	VAR robtarget Openhole_4144 := [[463.64, -19.43, 181.36], [0.050906, 0.705272, 0.70561, -0.045991], [0,0,0,0], [9E9, 9E9, 9E9, 9E9, 9E9, 9E9]];
	VAR robtarget Openhole_4145 := [[462.64, -19.54, 181.37], [0.047948, 0.705479, 0.70584, -0.042314], [0,0,0,0], [9E9, 9E9, 9E9, 9E9, 9E9, 9E9]];
	VAR robtarget Openhole_4146 := [[462.15, -19.58, 181.37], [0.046425, 0.705581, 0.705946, -0.040505], [0,0,0,0], [9E9, 9E9, 9E9, 9E9, 9E9, 9E9]];
	VAR robtarget Openhole_4147 := [[461.97, -18.21, 181.2], [0.041221, 0.705904, 0.705703, -0.044533], [0,0,0,0], [9E9, 9E9, 9E9, 9E9, 9E9, 9E9]];
	VAR robtarget Openhole_4148 := [[462.42, -18, 181.17], [0.042026, 0.705857, 0.705559, -0.046754], [0,0,0,0], [9E9, 9E9, 9E9, 9E9, 9E9, 9E9]];
	VAR robtarget Openhole_4149 := [[462.86, -17.76, 181.14], [0.042707, 0.705816, 0.705406, -0.049014], [0,0,0,0], [9E9, 9E9, 9E9, 9E9, 9E9, 9E9]];
	VAR robtarget Openhole_4150 := [[463.78, -17.37, 181.07], [0.044472, 0.705707, 0.705089, -0.05338], [0,0,0,0], [9E9, 9E9, 9E9, 9E9, 9E9, 9E9]];
	VAR robtarget Openhole_4151 := [[465.15, -16.77, 180.96], [0.046983, 0.705544, 0.704561, -0.059949], [0,0,0,0], [9E9, 9E9, 9E9, 9E9, 9E9, 9E9]];
	VAR robtarget Openhole_4152 := [[465.61, -16.58, 180.92], [0.047874, 0.705484, 0.704374, -0.062109], [0,0,0,0], [9E9, 9E9, 9E9, 9E9, 9E9, 9E9]];
	VAR robtarget Openhole_4153 := [[466.54, -16.21, 180.84], [0.049743, 0.705355, 0.703984, -0.066377], [0,0,0,0], [9E9, 9E9, 9E9, 9E9, 9E9, 9E9]];
	VAR robtarget Openhole_4154 := [[467.01, -16.05, 180.8], [0.050745, 0.705284, 0.703784, -0.068473], [0,0,0,0], [9E9, 9E9, 9E9, 9E9, 9E9, 9E9]];
	VAR robtarget Openhole_4155 := [[468.44, -15.62, 180.68], [0.054057, 0.705038, 0.703163, -0.074578], [0,0,0,0], [9E9, 9E9, 9E9, 9E9, 9E9, 9E9]];
	VAR robtarget Openhole_4156 := [[469.41, -15.37, 180.6], [0.056399, 0.704854, 0.702731, -0.078546], [0,0,0,0], [9E9, 9E9, 9E9, 9E9, 9E9, 9E9]];
	VAR robtarget Openhole_4157 := [[471.36, -14.97, 180.44], [0.061473, 0.70443, 0.701836, -0.086172], [0,0,0,0], [9E9, 9E9, 9E9, 9E9, 9E9, 9E9]];
	VAR robtarget Openhole_4158 := [[471.85, -14.89, 180.41], [0.062812, 0.704311, 0.701608, -0.088016], [0,0,0,0], [9E9, 9E9, 9E9, 9E9, 9E9, 9E9]];
	VAR robtarget Openhole_4159 := [[472.34, -14.82, 180.37], [0.064187, 0.704187, 0.701378, -0.089827], [0,0,0,0], [9E9, 9E9, 9E9, 9E9, 9E9, 9E9]];
	VAR robtarget Openhole_4160 := [[476.32, -14.47, 180.12], [0.075867, 0.703025, 0.699486, -0.103534], [0,0,0,0], [9E9, 9E9, 9E9, 9E9, 9E9, 9E9]];
	VAR robtarget Openhole_4161 := [[480.81, -14.37, 179.89], [0.089756, 0.701387, 0.697242, -0.1177], [0,0,0,0], [9E9, 9E9, 9E9, 9E9, 9E9, 9E9]];
	VAR robtarget Openhole_4162 := [[481.31, -14.37, 179.87], [0.091317, 0.701186, 0.696985, -0.119214], [0,0,0,0], [9E9, 9E9, 9E9, 9E9, 9E9, 9E9]];
	VAR robtarget Openhole_4163 := [[493.8, -14.52, 179.37], [0.129179, 0.695207, 0.68991, -0.154997], [0,0,0,0], [9E9, 9E9, 9E9, 9E9, 9E9, 9E9]];
	VAR robtarget Openhole_4164 := [[494.3, -14.52, 179.35], [0.130608, 0.69494, 0.689599, -0.156376], [0,0,0,0], [9E9, 9E9, 9E9, 9E9, 9E9, 9E9]];
	VAR robtarget Openhole_4165 := [[501.29, -14.35, 178.96], [0.14953, 0.691116, 0.684966, -0.17556], [0,0,0,0], [9E9, 9E9, 9E9, 9E9, 9E9, 9E9]];
	VAR robtarget Openhole_4166 := [[504.34, -14.15, 178.72], [0.157093, 0.689436, 0.682764, -0.18394], [0,0,0,0], [9E9, 9E9, 9E9, 9E9, 9E9, 9E9]];
	VAR robtarget Openhole_4167 := [[509.34, -14.15, 178.48], [0.183051, 0.683002, 0.683002, -0.183051], [0,0,0,0], [9E9, 9E9, 9E9, 9E9, 9E9, 9E9]];
	VAR robtarget Openhole_4168 := [[536.34, -14.15, 178.4], [0.183051, 0.683002, 0.683002, -0.183051], [0,0,0,0], [9E9, 9E9, 9E9, 9E9, 9E9, 9E9]];
	VAR robtarget Openhole_4169 := [[536.34, -15.36, 179.1], [0.183051, 0.683002, 0.683002, -0.183051], [0,0,0,0], [9E9, 9E9, 9E9, 9E9, 9E9, 9E9]];
	VAR robtarget Openhole_4170 := [[509.34, -15.36, 179.18], [0.183051, 0.683002, 0.683002, -0.183051], [0,0,0,0], [9E9, 9E9, 9E9, 9E9, 9E9, 9E9]];
	VAR robtarget Openhole_4171 := [[504.34, -15.36, 179.36], [0.160633, 0.68862, 0.683698, -0.180435], [0,0,0,0], [9E9, 9E9, 9E9, 9E9, 9E9, 9E9]];
	VAR robtarget Openhole_4172 := [[503.64, -15.39, 179.4], [0.158893, 0.689023, 0.684188, -0.17857], [0,0,0,0], [9E9, 9E9, 9E9, 9E9, 9E9, 9E9]];
	VAR robtarget Openhole_4173 := [[497.66, -15.67, 179.74], [0.143563, 0.69238, 0.68829, -0.16204], [0,0,0,0], [9E9, 9E9, 9E9, 9E9, 9E9, 9E9]];
	VAR robtarget Openhole_4174 := [[492.66, -15.73, 179.93], [0.129648, 0.69512, 0.691421, -0.148113], [0,0,0,0], [9E9, 9E9, 9E9, 9E9, 9E9, 9E9]];
	VAR robtarget Openhole_4175 := [[492.16, -15.73, 179.94], [0.128206, 0.695387, 0.69172, -0.14671], [0,0,0,0], [9E9, 9E9, 9E9, 9E9, 9E9, 9E9]];
	VAR robtarget Openhole_4176 := [[479.17, -15.58, 180.31], [0.08852, 0.701544, 0.698689, -0.108782], [0,0,0,0], [9E9, 9E9, 9E9, 9E9, 9E9, 9E9]];
	VAR robtarget Openhole_4177 := [[478.67, -15.58, 180.33], [0.086952, 0.70174, 0.698928, -0.107236], [0,0,0,0], [9E9, 9E9, 9E9, 9E9, 9E9, 9E9]];
	VAR robtarget Openhole_4178 := [[473.18, -15.79, 180.56], [0.070096, 0.703624, 0.701444, -0.089311], [0,0,0,0], [9E9, 9E9, 9E9, 9E9, 9E9, 9E9]];
	VAR robtarget Openhole_4179 := [[472.19, -15.88, 180.61], [0.06716, 0.70391, 0.701877, -0.085843], [0,0,0,0], [9E9, 9E9, 9E9, 9E9, 9E9, 9E9]];
	VAR robtarget Openhole_4180 := [[470.21, -16.14, 180.72], [0.061568, 0.704421, 0.702724, -0.078607], [0,0,0,0], [9E9, 9E9, 9E9, 9E9, 9E9, 9E9]];
	VAR robtarget Openhole_4181 := [[469.72, -16.22, 180.75], [0.060245, 0.704536, 0.702932, -0.076728], [0,0,0,0], [9E9, 9E9, 9E9, 9E9, 9E9, 9E9]];
	VAR robtarget Openhole_4182 := [[469.23, -16.32, 180.78], [0.058959, 0.704644, 0.703137, -0.074818], [0,0,0,0], [9E9, 9E9, 9E9, 9E9, 9E9, 9E9]];
	VAR robtarget Openhole_4183 := [[468.25, -16.53, 180.85], [0.056462, 0.704849, 0.70354, -0.070932], [0,0,0,0], [9E9, 9E9, 9E9, 9E9, 9E9, 9E9]];
	VAR robtarget Openhole_4184 := [[467.28, -16.77, 180.91], [0.054055, 0.705038, 0.703928, -0.06697], [0,0,0,0], [9E9, 9E9, 9E9, 9E9, 9E9, 9E9]];
	VAR robtarget Openhole_4185 := [[466.6, -18.47, 181.21], [0.05751, 0.704764, 0.704638, -0.059033], [0,0,0,0], [9E9, 9E9, 9E9, 9E9, 9E9, 9E9]];
	VAR robtarget Openhole_4186 := [[467.1, -18.42, 181.2], [0.058957, 0.704645, 0.704483, -0.060861], [0,0,0,0], [9E9, 9E9, 9E9, 9E9, 9E9, 9E9]];
	VAR robtarget Openhole_4187 := [[469.59, -18.24, 181.15], [0.066531, 0.70397, 0.70367, -0.069634], [0,0,0,0], [9E9, 9E9, 9E9, 9E9, 9E9, 9E9]];
	VAR robtarget Openhole_4188 := [[471.09, -18.16, 181.12], [0.071149, 0.703518, 0.703144, -0.074759], [0,0,0,0], [9E9, 9E9, 9E9, 9E9, 9E9, 9E9]];
	VAR robtarget Openhole_4189 := [[474.59, -18.11, 181.08], [0.082252, 0.702307, 0.701837, -0.086167], [0,0,0,0], [9E9, 9E9, 9E9, 9E9, 9E9, 9E9]];
	VAR robtarget Openhole_4190 := [[475.09, -18.11, 181.07], [0.083854, 0.702117, 0.701641, -0.087751], [0,0,0,0], [9E9, 9E9, 9E9, 9E9, 9E9, 9E9]];
	VAR robtarget Openhole_4191 := [[491.09, -18.34, 181.03], [0.133169, 0.694454, 0.693988, -0.135576], [0,0,0,0], [9E9, 9E9, 9E9, 9E9, 9E9, 9E9]];
	VAR robtarget Openhole_4192 := [[491.59, -18.34, 181.02], [0.134604, 0.694177, 0.693706, -0.137011], [0,0,0,0], [9E9, 9E9, 9E9, 9E9, 9E9, 9E9]];
	VAR robtarget Openhole_4193 := [[500.08, -18.17, 180.88], [0.157649, 0.689309, 0.68852, -0.16106], [0,0,0,0], [9E9, 9E9, 9E9, 9E9, 9E9, 9E9]];
	VAR robtarget Openhole_4194 := [[504.34, -17.96, 180.74], [0.168255, 0.686797, 0.685654, -0.172856], [0,0,0,0], [9E9, 9E9, 9E9, 9E9, 9E9, 9E9]];
	VAR robtarget Openhole_4195 := [[536.34, -17.96, 180.6], [0.183051, 0.683002, 0.683002, -0.183051], [0,0,0,0], [9E9, 9E9, 9E9, 9E9, 9E9, 9E9]];
	VAR robtarget Openhole_4196 := [[536.34, -17.24, 180.18], [0.183051, 0.683002, 0.683002, -0.183051], [0,0,0,0], [9E9, 9E9, 9E9, 9E9, 9E9, 9E9]];
	VAR robtarget Openhole_4197 := [[509.34, -17.24, 180.27], [0.183051, 0.683002, 0.683002, -0.183051], [0,0,0,0], [9E9, 9E9, 9E9, 9E9, 9E9, 9E9]];
	VAR robtarget Openhole_4198 := [[504.34, -17.24, 180.36], [0.166145, 0.687311, 0.68512, -0.174958], [0,0,0,0], [9E9, 9E9, 9E9, 9E9, 9E9, 9E9]];
	VAR robtarget Openhole_4199 := [[503.53, -17.27, 180.39], [0.16412, 0.687797, 0.685673, -0.172779], [0,0,0,0], [9E9, 9E9, 9E9, 9E9, 9E9, 9E9]];
	VAR robtarget Openhole_4200 := [[496.04, -17.57, 180.65], [0.144824, 0.692117, 0.690599, -0.151898], [0,0,0,0], [9E9, 9E9, 9E9, 9E9, 9E9, 9E9]];
	VAR robtarget Openhole_4201 := [[491.04, -17.63, 180.74], [0.130836, 0.694897, 0.693575, -0.13767], [0,0,0,0], [9E9, 9E9, 9E9, 9E9, 9E9, 9E9]];
	VAR robtarget Openhole_4202 := [[490.54, -17.62, 180.75], [0.12939, 0.695168, 0.693859, -0.136235], [0,0,0,0], [9E9, 9E9, 9E9, 9E9, 9E9, 9E9]];
	VAR robtarget Openhole_4203 := [[481.55, -17.51, 180.83], [0.102112, 0.699695, 0.698518, -0.109878], [0,0,0,0], [9E9, 9E9, 9E9, 9E9, 9E9, 9E9]];
	VAR robtarget Openhole_4204 := [[483.56, -27.51, 184.1], [0.140041, 0.693101, 0.702095, -0.084038], [0,0,0,0], [9E9, 9E9, 9E9, 9E9, 9E9, 9E9]];
	VAR robtarget Openhole_4205 := [[469.62, -28.25, 183.1], [0.099717, 0.70004, 0.706166, -0.036472], [0,0,0,0], [9E9, 9E9, 9E9, 9E9, 9E9, 9E9]];
	VAR robtarget Openhole_4206 := [[459.18, -29.01, 182.25], [0.068229, 0.703807, 0.707106, 0.001287], [0,0,0,0], [9E9, 9E9, 9E9, 9E9, 9E9, 9E9]];
	VAR robtarget Openhole_4207 := [[458.68, -29.06, 182.2], [0.066749, 0.703949, 0.7071, 0.003143], [0,0,0,0], [9E9, 9E9, 9E9, 9E9, 9E9, 9E9]];
	VAR robtarget Openhole_4208 := [[453.24, -29.67, 181.7], [0.050532, 0.705299, 0.706708, 0.023732], [0,0,0,0], [9E9, 9E9, 9E9, 9E9, 9E9, 9E9]];
	VAR robtarget Openhole_4209 := [[451.75, -29.75, 181.55], [0.045761, 0.705624, 0.706509, 0.029076], [0,0,0,0], [9E9, 9E9, 9E9, 9E9, 9E9, 9E9]];
	VAR robtarget Openhole_4210 := [[451.25, -29.75, 181.5], [0.044087, 0.705731, 0.706437, 0.030779], [0,0,0,0], [9E9, 9E9, 9E9, 9E9, 9E9, 9E9]];
	VAR robtarget Openhole_4211 := [[450.76, -29.75, 181.45], [0.042398, 0.705835, 0.706361, 0.032468], [0,0,0,0], [9E9, 9E9, 9E9, 9E9, 9E9, 9E9]];
	VAR robtarget Openhole_4212 := [[443.3, -29.47, 180.69], [0.016061, 0.706924, 0.704827, 0.056741], [0,0,0,0], [9E9, 9E9, 9E9, 9E9, 9E9, 9E9]];
	VAR robtarget Openhole_4213 := [[441.81, -29.49, 180.54], [0.011046, 0.707021, 0.7044, 0.061815], [0,0,0,0], [9E9, 9E9, 9E9, 9E9, 9E9, 9E9]];
	VAR robtarget Openhole_4214 := [[439.82, -29.61, 180.33], [0.004667, 0.707091, 0.703749, 0.068824], [0,0,0,0], [9E9, 9E9, 9E9, 9E9, 9E9, 9E9]];
	VAR robtarget Openhole_4215 := [[437.85, -29.84, 180.11], [-0.001273, 0.707106, 0.702996, 0.076135], [0,0,0,0], [9E9, 9E9, 9E9, 9E9, 9E9, 9E9]];
	VAR robtarget Openhole_4216 := [[428.05, -31.34, 178.78], [-0.029391, 0.706496, 0.698073, 0.112667], [0,0,0,0], [9E9, 9E9, 9E9, 9E9, 9E9, 9E9]];
	VAR robtarget Openhole_4217 := [[431.47, -29.27, 179.54], [-0.024758, 0.706673, 0.700692, 0.095033], [0,0,0,0], [9E9, 9E9, 9E9, 9E9, 9E9, 9E9]];
	VAR robtarget Openhole_4218 := [[437.75, -27.77, 180.33], [-0.008539, 0.707055, 0.703674, 0.069589], [0,0,0,0], [9E9, 9E9, 9E9, 9E9, 9E9, 9E9]];
	VAR robtarget Openhole_4219 := [[441.62, -26.84, 180.72], [0.001473, 0.707105, 0.705075, 0.053567], [0,0,0,0], [9E9, 9E9, 9E9, 9E9, 9E9, 9E9]];
	VAR robtarget Openhole_4220 := [[442.1, -26.73, 180.76], [0.002763, 0.707101, 0.705224, 0.051573], [0,0,0,0], [9E9, 9E9, 9E9, 9E9, 9E9, 9E9]];
	VAR robtarget Openhole_4221 := [[443.06, -26.45, 180.85], [0.005079, 0.707089, 0.705515, 0.04742], [0,0,0,0], [9E9, 9E9, 9E9, 9E9, 9E9, 9E9]];
	VAR robtarget Openhole_4222 := [[443.53, -26.29, 180.89], [0.006162, 0.70708, 0.705654, 0.045301], [0,0,0,0], [9E9, 9E9, 9E9, 9E9, 9E9, 9E9]];
	VAR robtarget Openhole_4223 := [[444.45, -25.91, 180.98], [0.008012, 0.707061, 0.705922, 0.040911], [0,0,0,0], [9E9, 9E9, 9E9, 9E9, 9E9, 9E9]];
	VAR robtarget Openhole_4224 := [[445.06, -25.46, 181.04], [0.008543, 0.707055, 0.706122, 0.037314], [0,0,0,0], [9E9, 9E9, 9E9, 9E9, 9E9, 9E9]];
	VAR robtarget Openhole_4225 := [[442.67, -23.11, 181.04], [-0.007574, 0.707066, 0.706114, 0.037453], [0,0,0,0], [9E9, 9E9, 9E9, 9E9, 9E9, 9E9]];
	VAR robtarget Openhole_4226 := [[442.05, -23.57, 180.98], [-0.008101, 0.70706, 0.705912, 0.041093], [0,0,0,0], [9E9, 9E9, 9E9, 9E9, 9E9, 9E9]];
	VAR robtarget Openhole_4227 := [[441.65, -23.86, 180.94], [-0.008486, 0.707056, 0.705771, 0.043439], [0,0,0,0], [9E9, 9E9, 9E9, 9E9, 9E9, 9E9]];
	VAR robtarget Openhole_4228 := [[441.23, -24.14, 180.9], [-0.008974, 0.70705, 0.705624, 0.045762], [0,0,0,0], [9E9, 9E9, 9E9, 9E9, 9E9, 9E9]];
	VAR robtarget Openhole_4229 := [[440.8, -24.39, 180.86], [-0.009587, 0.707042, 0.705472, 0.048053], [0,0,0,0], [9E9, 9E9, 9E9, 9E9, 9E9, 9E9]];
	VAR robtarget Openhole_4230 := [[439.91, -24.83, 180.77], [-0.011121, 0.707019, 0.705153, 0.052533], [0,0,0,0], [9E9, 9E9, 9E9, 9E9, 9E9, 9E9]];
	VAR robtarget Openhole_4231 := [[439.46, -25.04, 180.73], [-0.011943, 0.707006, 0.704984, 0.05475], [0,0,0,0], [9E9, 9E9, 9E9, 9E9, 9E9, 9E9]];
	VAR robtarget Openhole_4232 := [[438.55, -25.44, 180.63], [-0.013681, 0.706974, 0.70463, 0.059135], [0,0,0,0], [9E9, 9E9, 9E9, 9E9, 9E9, 9E9]];
	VAR robtarget Openhole_4233 := [[434.35, -26.98, 180.15], [-0.022715, 0.706742, 0.702776, 0.078142], [0,0,0,0], [9E9, 9E9, 9E9, 9E9, 9E9, 9E9]];
	VAR robtarget Openhole_4234 := [[432.92, -27.42, 179.98], [-0.026057, 0.706627, 0.702072, 0.08423], [0,0,0,0], [9E9, 9E9, 9E9, 9E9, 9E9, 9E9]];
	VAR robtarget Openhole_4235 := [[435.85, -24.75, 180.56], [-0.025139, 0.70666, 0.704043, 0.065752], [0,0,0,0], [9E9, 9E9, 9E9, 9E9, 9E9, 9E9]];
	VAR robtarget Openhole_4236 := [[437.63, -23.85, 180.76], [-0.022173, 0.706759, 0.704818, 0.056851], [0,0,0,0], [9E9, 9E9, 9E9, 9E9, 9E9, 9E9]];
	VAR robtarget Openhole_4237 := [[438.06, -23.61, 180.8], [-0.021498, 0.70678, 0.704996, 0.054595], [0,0,0,0], [9E9, 9E9, 9E9, 9E9, 9E9, 9E9]];
	VAR robtarget Openhole_4238 := [[439.34, -22.84, 180.93], [-0.019787, 0.70683, 0.705495, 0.04772], [0,0,0,0], [9E9, 9E9, 9E9, 9E9, 9E9, 9E9]];
	VAR robtarget Openhole_4239 := [[440.59, -22.01, 181.05], [-0.018371, 0.706868, 0.705932, 0.040747], [0,0,0,0], [9E9, 9E9, 9E9, 9E9, 9E9, 9E9]];
	VAR robtarget Openhole_4240 := [[441.01, -21.74, 181.08], [-0.017863, 0.706881, 0.706062, 0.038424], [0,0,0,0], [9E9, 9E9, 9E9, 9E9, 9E9, 9E9]];
	VAR robtarget Openhole_4241 := [[441.8, -21.35, 181.13], [-0.016509, 0.706914, 0.706268, 0.03444], [0,0,0,0], [9E9, 9E9, 9E9, 9E9, 9E9, 9E9]];
	VAR robtarget Openhole_4242 := [[438.17, -20.01, 181.2], [-0.033312, 0.706322, 0.705852, 0.042112], [0,0,0,0], [9E9, 9E9, 9E9, 9E9, 9E9, 9E9]];
	VAR robtarget Openhole_4243 := [[437.76, -20.3, 181.16], [-0.033719, 0.706302, 0.705709, 0.044445], [0,0,0,0], [9E9, 9E9, 9E9, 9E9, 9E9, 9E9]];
	VAR robtarget Openhole_4244 := [[436.96, -20.89, 181.08], [-0.034413, 0.706269, 0.705399, 0.049119], [0,0,0,0], [9E9, 9E9, 9E9, 9E9, 9E9, 9E9]];
	VAR robtarget Openhole_4245 := [[436.14, -21.45, 180.99], [-0.035276, 0.706226, 0.705061, 0.053749], [0,0,0,0], [9E9, 9E9, 9E9, 9E9, 9E9, 9E9]];
	VAR robtarget Openhole_4246 := [[435.72, -21.72, 180.95], [-0.035777, 0.706201, 0.704882, 0.056046], [0,0,0,0], [9E9, 9E9, 9E9, 9E9, 9E9, 9E9]];
	VAR robtarget Openhole_4247 := [[435.29, -21.98, 180.9], [-0.03632, 0.706173, 0.704697, 0.058327], [0,0,0,0], [9E9, 9E9, 9E9, 9E9, 9E9, 9E9]];
	VAR robtarget Openhole_4248 := [[434.43, -22.48, 180.81], [-0.037528, 0.70611, 0.704308, 0.062847], [0,0,0,0], [9E9, 9E9, 9E9, 9E9, 9E9, 9E9]];
	VAR robtarget Openhole_4249 := [[434, -22.72, 180.76], [-0.038199, 0.706074, 0.704105, 0.065082], [0,0,0,0], [9E9, 9E9, 9E9, 9E9, 9E9, 9E9]];
	VAR robtarget Openhole_4250 := [[433.55, -22.94, 180.71], [-0.038932, 0.706034, 0.703898, 0.067292], [0,0,0,0], [9E9, 9E9, 9E9, 9E9, 9E9, 9E9]];
	VAR robtarget Openhole_4251 := [[432.65, -23.37, 180.6], [-0.040522, 0.705945, 0.703467, 0.071658], [0,0,0,0], [9E9, 9E9, 9E9, 9E9, 9E9, 9E9]];
	VAR robtarget Openhole_4252 := [[432.19, -23.56, 180.55], [-0.041401, 0.705894, 0.703245, 0.0738], [0,0,0,0], [9E9, 9E9, 9E9, 9E9, 9E9, 9E9]];
	VAR robtarget Openhole_4253 := [[431.73, -23.75, 180.5], [-0.042318, 0.705839, 0.703019, 0.075923], [0,0,0,0], [9E9, 9E9, 9E9, 9E9, 9E9, 9E9]];
	VAR robtarget Openhole_4254 := [[430.8, -24.09, 180.4], [-0.044272, 0.705719, 0.702555, 0.0801], [0,0,0,0], [9E9, 9E9, 9E9, 9E9, 9E9, 9E9]];
	VAR robtarget Openhole_4255 := [[430.33, -24.25, 180.35], [-0.045321, 0.705653, 0.702319, 0.082146], [0,0,0,0], [9E9, 9E9, 9E9, 9E9, 9E9, 9E9]];
	VAR robtarget Openhole_4256 := [[427.45, -25.03, 180.04], [-0.052266, 0.705173, 0.700837, 0.093957], [0,0,0,0], [9E9, 9E9, 9E9, 9E9, 9E9, 9E9]];
	VAR robtarget Openhole_4257 := [[426.96, -25.13, 179.99], [-0.053519, 0.705079, 0.700581, 0.095848], [0,0,0,0], [9E9, 9E9, 9E9, 9E9, 9E9, 9E9]];
	VAR robtarget Openhole_4258 := [[425, -25.46, 179.79], [-0.058849, 0.704654, 0.699545, 0.103137], [0,0,0,0], [9E9, 9E9, 9E9, 9E9, 9E9, 9E9]];
	VAR robtarget Openhole_4259 := [[421.03, -25.86, 179.44], [-0.070416, 0.703592, 0.69741, 0.1167], [0,0,0,0], [9E9, 9E9, 9E9, 9E9, 9E9, 9E9]];
	VAR robtarget Openhole_4260 := [[416.05, -25.98, 179.07], [-0.085851, 0.701876, 0.694657, 0.132106], [0,0,0,0], [9E9, 9E9, 9E9, 9E9, 9E9, 9E9]];
	VAR robtarget Openhole_4261 := [[415.55, -25.97, 179.04], [-0.087426, 0.701681, 0.694377, 0.133569], [0,0,0,0], [9E9, 9E9, 9E9, 9E9, 9E9, 9E9]];
	VAR robtarget Openhole_4262 := [[401.58, -25.68, 178.24], [-0.130137, 0.695028, 0.685922, 0.171786], [0,0,0,0], [9E9, 9E9, 9E9, 9E9, 9E9, 9E9]];
	VAR robtarget Openhole_4263 := [[401.08, -25.68, 178.21], [-0.131554, 0.694762, 0.685591, 0.173103], [0,0,0,0], [9E9, 9E9, 9E9, 9E9, 9E9, 9E9]];
	VAR robtarget Openhole_4264 := [[395.6, -25.83, 177.78], [-0.146298, 0.691807, 0.681759, 0.187629], [0,0,0,0], [9E9, 9E9, 9E9, 9E9, 9E9, 9E9]];
	VAR robtarget Openhole_4265 := [[395.1, -25.86, 177.73], [-0.147556, 0.69154, 0.681393, 0.188956], [0,0,0,0], [9E9, 9E9, 9E9, 9E9, 9E9, 9E9]];
	VAR robtarget Openhole_4266 := [[394.33, -25.89, 177.67], [-0.149558, 0.69111, 0.680843, 0.190928], [0,0,0,0], [9E9, 9E9, 9E9, 9E9, 9E9, 9E9]];
	VAR robtarget Openhole_4267 := [[389.33, -25.89, 177.34], [-0.162718, 0.68813, 0.677341, 0.203], [0,0,0,0], [9E9, 9E9, 9E9, 9E9, 9E9, 9E9]];
	VAR robtarget Openhole_4268 := [[362.33, -25.89, 177.42], [-0.183051, 0.683002, 0.683002, 0.183051], [0,0,0,0], [9E9, 9E9, 9E9, 9E9, 9E9, 9E9]];
	VAR robtarget Openhole_4269 := [[362.33, -25.1, 177.88], [-0.183051, 0.683002, 0.683002, 0.183051], [0,0,0,0], [9E9, 9E9, 9E9, 9E9, 9E9, 9E9]];
	VAR robtarget Openhole_4270 := [[389.33, -25.1, 177.79], [-0.164965, 0.687595, 0.678001, 0.200786], [0,0,0,0], [9E9, 9E9, 9E9, 9E9, 9E9, 9E9]];
	VAR robtarget Openhole_4271 := [[394.34, -25.1, 178.09], [-0.151861, 0.690607, 0.681475, 0.188657], [0,0,0,0], [9E9, 9E9, 9E9, 9E9, 9E9, 9E9]];
	VAR robtarget Openhole_4272 := [[395.22, -25.08, 178.15], [-0.149548, 0.691112, 0.682101, 0.18638], [0,0,0,0], [9E9, 9E9, 9E9, 9E9, 9E9, 9E9]];
	VAR robtarget Openhole_4273 := [[400.7, -24.87, 178.57], [-0.135064, 0.694088, 0.685946, 0.171692], [0,0,0,0], [9E9, 9E9, 9E9, 9E9, 9E9, 9E9]];
	VAR robtarget Openhole_4274 := [[402.2, -24.86, 178.65], [-0.130856, 0.694893, 0.686935, 0.16769], [0,0,0,0], [9E9, 9E9, 9E9, 9E9, 9E9, 9E9]];
	VAR robtarget Openhole_4275 := [[402.7, -24.86, 178.68], [-0.129427, 0.695161, 0.687259, 0.166358], [0,0,0,0], [9E9, 9E9, 9E9, 9E9, 9E9, 9E9]];
	VAR robtarget Openhole_4276 := [[416.18, -25.08, 179.37], [-0.088322, 0.701569, 0.69526, 0.128891], [0,0,0,0], [9E9, 9E9, 9E9, 9E9, 9E9, 9E9]];
	VAR robtarget Openhole_4277 := [[416.68, -25.08, 179.4], [-0.086764, 0.701764, 0.695535, 0.127399], [0,0,0,0], [9E9, 9E9, 9E9, 9E9, 9E9, 9E9]];
	VAR robtarget Openhole_4278 := [[422.16, -24.91, 179.76], [-0.069892, 0.703644, 0.698473, 0.110163], [0,0,0,0], [9E9, 9E9, 9E9, 9E9, 9E9, 9E9]];
	VAR robtarget Openhole_4279 := [[424.15, -24.72, 179.92], [-0.064077, 0.704198, 0.699509, 0.103381], [0,0,0,0], [9E9, 9E9, 9E9, 9E9, 9E9, 9E9]];
	VAR robtarget Openhole_4280 := [[425.13, -24.59, 180], [-0.06127, 0.704447, 0.700019, 0.099868], [0,0,0,0], [9E9, 9E9, 9E9, 9E9, 9E9, 9E9]];
	VAR robtarget Openhole_4281 := [[426.61, -24.36, 180.13], [-0.05721, 0.704789, 0.700772, 0.094438], [0,0,0,0], [9E9, 9E9, 9E9, 9E9, 9E9, 9E9]];
	VAR robtarget Openhole_4282 := [[427.1, -24.27, 180.18], [-0.055917, 0.704892, 0.701021, 0.092573], [0,0,0,0], [9E9, 9E9, 9E9, 9E9, 9E9, 9E9]];
	VAR robtarget Openhole_4283 := [[428.07, -24.05, 180.27], [-0.053429, 0.705085, 0.701514, 0.088762], [0,0,0,0], [9E9, 9E9, 9E9, 9E9, 9E9, 9E9]];
	VAR robtarget Openhole_4284 := [[429.52, -23.69, 180.41], [-0.049857, 0.705347, 0.70223, 0.082903], [0,0,0,0], [9E9, 9E9, 9E9, 9E9, 9E9, 9E9]];
	VAR robtarget Openhole_4285 := [[430.48, -23.42, 180.5], [-0.047597, 0.705503, 0.702691, 0.0789], [0,0,0,0], [9E9, 9E9, 9E9, 9E9, 9E9, 9E9]];
	VAR robtarget Openhole_4286 := [[428.63, -22.36, 180.64], [-0.057235, 0.704787, 0.70241, 0.081368], [0,0,0,0], [9E9, 9E9, 9E9, 9E9, 9E9, 9E9]];
	VAR robtarget Openhole_4287 := [[428.14, -22.45, 180.6], [-0.058526, 0.704681, 0.702188, 0.08326], [0,0,0,0], [9E9, 9E9, 9E9, 9E9, 9E9, 9E9]];
	VAR robtarget Openhole_4288 := [[425.18, -22.88, 180.4], [-0.06678, 0.703946, 0.700814, 0.094127], [0,0,0,0], [9E9, 9E9, 9E9, 9E9, 9E9, 9E9]];
	VAR robtarget Openhole_4289 := [[420.7, -23.18, 180.16], [-0.080232, 0.70254, 0.69864, 0.109096], [0,0,0,0], [9E9, 9E9, 9E9, 9E9, 9E9, 9E9]];
	VAR robtarget Openhole_4290 := [[418.2, -23.21, 180.05], [-0.088029, 0.701606, 0.697387, 0.116841], [0,0,0,0], [9E9, 9E9, 9E9, 9E9, 9E9, 9E9]];
	VAR robtarget Openhole_4291 := [[417.7, -23.21, 180.03], [-0.089597, 0.701407, 0.697131, 0.118355], [0,0,0,0], [9E9, 9E9, 9E9, 9E9, 9E9, 9E9]];
	VAR robtarget Openhole_4292 := [[417.2, -23.21, 180.01], [-0.091157, 0.701206, 0.696873, 0.119868], [0,0,0,0], [9E9, 9E9, 9E9, 9E9, 9E9, 9E9]];
	VAR robtarget Openhole_4293 := [[416.7, -23.21, 179.99], [-0.092728, 0.701, 0.696614, 0.121361], [0,0,0,0], [9E9, 9E9, 9E9, 9E9, 9E9, 9E9]];
	VAR robtarget Openhole_4294 := [[404.71, -23.06, 179.57], [-0.129184, 0.695206, 0.689809, 0.155447], [0,0,0,0], [9E9, 9E9, 9E9, 9E9, 9E9, 9E9]];
	VAR robtarget Openhole_4295 := [[404.21, -23.06, 179.55], [-0.130617, 0.694938, 0.689498, 0.15682], [0,0,0,0], [9E9, 9E9, 9E9, 9E9, 9E9, 9E9]];
	VAR robtarget Openhole_4296 := [[397.22, -23.22, 179.2], [-0.149636, 0.691093, 0.684882, 0.175887], [0,0,0,0], [9E9, 9E9, 9E9, 9E9, 9E9, 9E9]];
	VAR robtarget Openhole_4297 := [[395.23, -23.34, 179.06], [-0.154658, 0.689986, 0.683467, 0.18131], [0,0,0,0], [9E9, 9E9, 9E9, 9E9, 9E9, 9E9]];
	VAR robtarget Openhole_4298 := [[394.34, -23.36, 179.01], [-0.15695, 0.689468, 0.682848, 0.183626], [0,0,0,0], [9E9, 9E9, 9E9, 9E9, 9E9, 9E9]];
	VAR robtarget Openhole_4299 := [[389.34, -23.36, 178.8], [-0.169929, 0.686385, 0.679434, 0.195881], [0,0,0,0], [9E9, 9E9, 9E9, 9E9, 9E9, 9E9]];
	VAR robtarget Openhole_4300 := [[362.34, -23.36, 178.88], [-0.183051, 0.683002, 0.683002, 0.183051], [0,0,0,0], [9E9, 9E9, 9E9, 9E9, 9E9, 9E9]];
	VAR robtarget Openhole_4301 := [[362.34, -22.46, 179.4], [-0.183051, 0.683002, 0.683002, 0.183051], [0,0,0,0], [9E9, 9E9, 9E9, 9E9, 9E9, 9E9]];
	VAR robtarget Openhole_4302 := [[389.34, -22.46, 179.32], [-0.172507, 0.685741, 0.680165, 0.193326], [0,0,0,0], [9E9, 9E9, 9E9, 9E9, 9E9, 9E9]];
	VAR robtarget Openhole_4303 := [[394.34, -22.46, 179.48], [-0.159593, 0.688862, 0.683547, 0.181006], [0,0,0,0], [9E9, 9E9, 9E9, 9E9, 9E9, 9E9]];
	VAR robtarget Openhole_4304 := [[395.12, -22.43, 179.52], [-0.157612, 0.689317, 0.68409, 0.178945], [0,0,0,0], [9E9, 9E9, 9E9, 9E9, 9E9, 9E9]];
	VAR robtarget Openhole_4305 := [[401.61, -22.16, 179.86], [-0.140733, 0.692961, 0.688493, 0.161175], [0,0,0,0], [9E9, 9E9, 9E9, 9E9, 9E9, 9E9]];
	VAR robtarget Openhole_4306 := [[405.6, -22.12, 180], [-0.129492, 0.695149, 0.69099, 0.15011], [0,0,0,0], [9E9, 9E9, 9E9, 9E9, 9E9, 9E9]];
	VAR robtarget Openhole_4307 := [[406.1, -22.12, 180.01], [-0.128047, 0.695416, 0.691291, 0.148717], [0,0,0,0], [9E9, 9E9, 9E9, 9E9, 9E9, 9E9]];
	VAR robtarget Openhole_4308 := [[418.1, -22.26, 180.33], [-0.091403, 0.701174, 0.697838, 0.114113], [0,0,0,0], [9E9, 9E9, 9E9, 9E9, 9E9, 9E9]];
	VAR robtarget Openhole_4309 := [[418.6, -22.26, 180.34], [-0.089837, 0.701377, 0.698086, 0.112588], [0,0,0,0], [9E9, 9E9, 9E9, 9E9, 9E9, 9E9]];
	VAR robtarget Openhole_4310 := [[423.09, -22.18, 180.5], [-0.075824, 0.70303, 0.700227, 0.098401], [0,0,0,0], [9E9, 9E9, 9E9, 9E9, 9E9, 9E9]];
	VAR robtarget Openhole_4311 := [[427.57, -21.76, 180.73], [-0.062702, 0.704321, 0.70224, 0.082818], [0,0,0,0], [9E9, 9E9, 9E9, 9E9, 9E9, 9E9]];
	VAR robtarget Openhole_4312 := [[428.06, -21.68, 180.76], [-0.061338, 0.704441, 0.702454, 0.080981], [0,0,0,0], [9E9, 9E9, 9E9, 9E9, 9E9, 9E9]];
	VAR robtarget Openhole_4313 := [[429.04, -21.5, 180.82], [-0.058712, 0.704665, 0.702878, 0.077215], [0,0,0,0], [9E9, 9E9, 9E9, 9E9, 9E9, 9E9]];
	VAR robtarget Openhole_4314 := [[430.02, -21.29, 180.88], [-0.056228, 0.704868, 0.703294, 0.073334], [0,0,0,0], [9E9, 9E9, 9E9, 9E9, 9E9, 9E9]];
	VAR robtarget Openhole_4315 := [[432.43, -20.64, 181.04], [-0.05041, 0.705308, 0.704267, 0.063304], [0,0,0,0], [9E9, 9E9, 9E9, 9E9, 9E9, 9E9]];
	VAR robtarget Openhole_4316 := [[433.85, -20.18, 181.13], [-0.047219, 0.705528, 0.704801, 0.057064], [0,0,0,0], [9E9, 9E9, 9E9, 9E9, 9E9, 9E9]];
	VAR robtarget Openhole_4317 := [[434.32, -20.01, 181.16], [-0.046242, 0.705593, 0.70497, 0.054933], [0,0,0,0], [9E9, 9E9, 9E9, 9E9, 9E9, 9E9]];
	VAR robtarget Openhole_4318 := [[434.78, -19.82, 181.19], [-0.045338, 0.705652, 0.705135, 0.052766], [0,0,0,0], [9E9, 9E9, 9E9, 9E9, 9E9, 9E9]];
	VAR robtarget Openhole_4319 := [[435.69, -19.42, 181.25], [-0.043639, 0.705759, 0.70545, 0.048377], [0,0,0,0], [9E9, 9E9, 9E9, 9E9, 9E9, 9E9]];
	VAR robtarget Openhole_4320 := [[436.63, -19.07, 181.3], [-0.041667, 0.705878, 0.705731, 0.044086], [0,0,0,0], [9E9, 9E9, 9E9, 9E9, 9E9, 9E9]];
	VAR robtarget Openhole_4321 := [[437.08, -18.86, 181.32], [-0.040877, 0.705924, 0.705867, 0.041856], [0,0,0,0], [9E9, 9E9, 9E9, 9E9, 9E9, 9E9]];
	VAR robtarget Openhole_4322 := [[436.54, -17.57, 181.48], [-0.047034, 0.705541, 0.706011, 0.039358], [0,0,0,0], [9E9, 9E9, 9E9, 9E9, 9E9, 9E9]];
	VAR robtarget Openhole_4323 := [[435.54, -17.56, 181.5], [-0.050402, 0.705308, 0.705818, 0.042672], [0,0,0,0], [9E9, 9E9, 9E9, 9E9, 9E9, 9E9]];
	VAR robtarget Openhole_4324 := [[435.04, -17.58, 181.5], [-0.052004, 0.705192, 0.705711, 0.044402], [0,0,0,0], [9E9, 9E9, 9E9, 9E9, 9E9, 9E9]];
	VAR robtarget Openhole_4325 := [[434.54, -17.58, 181.51], [-0.053671, 0.705067, 0.705605, 0.046065], [0,0,0,0], [9E9, 9E9, 9E9, 9E9, 9E9, 9E9]];
	VAR robtarget Openhole_4326 := [[434.04, -17.59, 181.51], [-0.05532, 0.70494, 0.705493, 0.047741], [0,0,0,0], [9E9, 9E9, 9E9, 9E9, 9E9, 9E9]];
	VAR robtarget Openhole_4327 := [[433.54, -17.58, 181.52], [-0.057005, 0.704805, 0.705381, 0.049374], [0,0,0,0], [9E9, 9E9, 9E9, 9E9, 9E9, 9E9]];
	VAR robtarget Openhole_4328 := [[433.04, -17.58, 181.53], [-0.05864, 0.704671, 0.705261, 0.051054], [0,0,0,0], [9E9, 9E9, 9E9, 9E9, 9E9, 9E9]];
	VAR robtarget Openhole_4329 := [[432.54, -17.58, 181.53], [-0.060296, 0.704531, 0.70514, 0.052705], [0,0,0,0], [9E9, 9E9, 9E9, 9E9, 9E9, 9E9]];
	VAR robtarget Openhole_4330 := [[418.04, -17.3, 181.82], [-0.107598, 0.698872, 0.700238, 0.09832], [0,0,0,0], [9E9, 9E9, 9E9, 9E9, 9E9, 9E9]];
	VAR robtarget Openhole_4331 := [[408.55, -17.2, 182.02], [-0.136262, 0.693853, 0.695692, 0.126539], [0,0,0,0], [9E9, 9E9, 9E9, 9E9, 9E9, 9E9]];
	VAR robtarget Openhole_4332 := [[408.05, -17.2, 182.03], [-0.137698, 0.69357, 0.695426, 0.127996], [0,0,0,0], [9E9, 9E9, 9E9, 9E9, 9E9, 9E9]];
	VAR robtarget Openhole_4333 := [[398.55, -17.4, 182.1], [-0.163408, 0.687966, 0.689876, 0.155147], [0,0,0,0], [9E9, 9E9, 9E9, 9E9, 9E9, 9E9]];
	VAR robtarget Openhole_4334 := [[394.35, -17.6, 182.06], [-0.17381, 0.685412, 0.687145, 0.166826], [0,0,0,0], [9E9, 9E9, 9E9, 9E9, 9E9, 9E9]];
	VAR robtarget Openhole_4335 := [[362.35, -17.6, 182.21], [-0.183051, 0.683002, 0.683002, 0.183051], [0,0,0,0], [9E9, 9E9, 9E9, 9E9, 9E9, 9E9]];
	VAR robtarget Openhole_4336 := [[362.35, -18.56, 181.66], [-0.183051, 0.683002, 0.683002, 0.183051], [0,0,0,0], [9E9, 9E9, 9E9, 9E9, 9E9, 9E9]];
	VAR robtarget Openhole_4337 := [[389.35, -18.56, 181.57], [-0.183637, 0.682845, 0.68322, 0.182237], [0,0,0,0], [9E9, 9E9, 9E9, 9E9, 9E9, 9E9]];
	VAR robtarget Openhole_4338 := [[394.35, -18.56, 181.55], [-0.171006, 0.686117, 0.686458, 0.169635], [0,0,0,0], [9E9, 9E9, 9E9, 9E9, 9E9, 9E9]];
	VAR robtarget Openhole_4339 := [[402.43, -18.22, 181.66], [-0.150382, 0.690931, 0.691649, 0.147044], [0,0,0,0], [9E9, 9E9, 9E9, 9E9, 9E9, 9E9]];
	VAR robtarget Openhole_4340 := [[408.43, -18.16, 181.64], [-0.133611, 0.694369, 0.695081, 0.129855], [0,0,0,0], [9E9, 9E9, 9E9, 9E9, 9E9, 9E9]];
	VAR robtarget Openhole_4341 := [[408.93, -18.16, 181.64], [-0.132157, 0.694647, 0.69535, 0.128408], [0,0,0,0], [9E9, 9E9, 9E9, 9E9, 9E9, 9E9]];
	VAR robtarget Openhole_4342 := [[426.43, -18.45, 181.43], [-0.077393, 0.702859, 0.70306, 0.075543], [0,0,0,0], [9E9, 9E9, 9E9, 9E9, 9E9, 9E9]];
	VAR robtarget Openhole_4343 := [[426.93, -18.44, 181.43], [-0.075782, 0.703034, 0.703232, 0.073923], [0,0,0,0], [9E9, 9E9, 9E9, 9E9, 9E9, 9E9]];
	VAR robtarget Openhole_4344 := [[430.43, -18.38, 181.42], [-0.064572, 0.704152, 0.704354, 0.062333], [0,0,0,0], [9E9, 9E9, 9E9, 9E9, 9E9, 9E9]];
	VAR robtarget Openhole_4345 := [[431.43, -18.38, 181.41], [-0.061279, 0.704446, 0.704637, 0.059052], [0,0,0,0], [9E9, 9E9, 9E9, 9E9, 9E9, 9E9]];
	VAR robtarget Openhole_4346 := [[431.92, -18.36, 181.41], [-0.05973, 0.70458, 0.704781, 0.05731], [0,0,0,0], [9E9, 9E9, 9E9, 9E9, 9E9, 9E9]];
	VAR robtarget Openhole_4347 := [[433.09, -19.64, 181.21], [-0.05156, 0.705224, 0.704744, 0.057758], [0,0,0,0], [9E9, 9E9, 9E9, 9E9, 9E9, 9E9]];
	VAR robtarget Openhole_4348 := [[431.14, -20.07, 181.12], [-0.056576, 0.70484, 0.704056, 0.065617], [0,0,0,0], [9E9, 9E9, 9E9, 9E9, 9E9, 9E9]];
	VAR robtarget Openhole_4349 := [[429.67, -20.35, 181.05], [-0.060491, 0.704515, 0.703497, 0.071356], [0,0,0,0], [9E9, 9E9, 9E9, 9E9, 9E9, 9E9]];
	VAR robtarget Openhole_4350 := [[429.17, -20.43, 181.03], [-0.061856, 0.704396, 0.703306, 0.073216], [0,0,0,0], [9E9, 9E9, 9E9, 9E9, 9E9, 9E9]];
	VAR robtarget Openhole_4351 := [[428.18, -20.56, 180.99], [-0.064676, 0.704143, 0.702918, 0.076851], [0,0,0,0], [9E9, 9E9, 9E9, 9E9, 9E9, 9E9]];
	VAR robtarget Openhole_4352 := [[426.19, -20.74, 180.92], [-0.070564, 0.703577, 0.702118, 0.08385], [0,0,0,0], [9E9, 9E9, 9E9, 9E9, 9E9, 9E9]];
	VAR robtarget Openhole_4353 := [[425.2, -20.8, 180.89], [-0.073579, 0.703268, 0.701704, 0.087248], [0,0,0,0], [9E9, 9E9, 9E9, 9E9, 9E9, 9E9]];
	VAR robtarget Openhole_4354 := [[421.2, -20.9, 180.79], [-0.086071, 0.701849, 0.699979, 0.100146], [0,0,0,0], [9E9, 9E9, 9E9, 9E9, 9E9, 9E9]];
	VAR robtarget Openhole_4355 := [[420.7, -20.89, 180.79], [-0.08766, 0.701652, 0.699756, 0.101695], [0,0,0,0], [9E9, 9E9, 9E9, 9E9, 9E9, 9E9]];
	VAR robtarget Openhole_4356 := [[406.7, -20.73, 180.6], [-0.130632, 0.694935, 0.692548, 0.142751], [0,0,0,0], [9E9, 9E9, 9E9, 9E9, 9E9, 9E9]];
	VAR robtarget Openhole_4357 := [[406.2, -20.73, 180.6], [-0.132071, 0.694663, 0.692255, 0.144164], [0,0,0,0], [9E9, 9E9, 9E9, 9E9, 9E9, 9E9]];
	VAR robtarget Openhole_4358 := [[398.21, -20.89, 180.38], [-0.153904, 0.690155, 0.687239, 0.16644], [0,0,0,0], [9E9, 9E9, 9E9, 9E9, 9E9, 9E9]];
	VAR robtarget Openhole_4359 := [[395.21, -21.06, 180.24], [-0.161406, 0.688439, 0.685186, 0.174702], [0,0,0,0], [9E9, 9E9, 9E9, 9E9, 9E9, 9E9]];
	VAR robtarget Openhole_4360 := [[394.34, -21.09, 180.21], [-0.163604, 0.68792, 0.68459, 0.17702], [0,0,0,0], [9E9, 9E9, 9E9, 9E9, 9E9, 9E9]];
	VAR robtarget Openhole_4361 := [[389.34, -21.09, 180.11], [-0.17642, 0.684745, 0.681258, 0.189439], [0,0,0,0], [9E9, 9E9, 9E9, 9E9, 9E9, 9E9]];
	VAR robtarget Openhole_4362 := [[362.34, -21.09, 180.19], [-0.183051, 0.683002, 0.683002, 0.183051], [0,0,0,0], [9E9, 9E9, 9E9, 9E9, 9E9, 9E9]];
	VAR robtarget Openhole_4363 := [[362.35, -15.88, 183.21], [-0.183051, 0.683002, 0.683002, 0.183051], [0,0,0,0], [9E9, 9E9, 9E9, 9E9, 9E9, 9E9]];
	VAR robtarget Openhole_4364 := [[389.35, -15.88, 183.12], [-0.19126, 0.680749, 0.685215, 0.174586], [0,0,0,0], [9E9, 9E9, 9E9, 9E9, 9E9, 9E9]];
	VAR robtarget Openhole_4365 := [[394.35, -15.88, 182.97], [-0.178824, 0.684121, 0.688349, 0.161791], [0,0,0,0], [9E9, 9E9, 9E9, 9E9, 9E9, 9E9]];
	VAR robtarget Openhole_4366 := [[402.84, -15.53, 182.87], [-0.157416, 0.689362, 0.693565, 0.137722], [0,0,0,0], [9E9, 9E9, 9E9, 9E9, 9E9, 9E9]];
	VAR robtarget Openhole_4367 := [[411.34, -15.42, 182.62], [-0.133709, 0.69435, 0.698062, 0.112734], [0,0,0,0], [9E9, 9E9, 9E9, 9E9, 9E9, 9E9]];
	VAR robtarget Openhole_4368 := [[411.84, -15.42, 182.6], [-0.132245, 0.69463, 0.698302, 0.111238], [0,0,0,0], [9E9, 9E9, 9E9, 9E9, 9E9, 9E9]];
	VAR robtarget Openhole_4369 := [[425.83, -15.62, 182.07], [-0.088646, 0.701528, 0.703814, 0.068159], [0,0,0,0], [9E9, 9E9, 9E9, 9E9, 9E9, 9E9]];
	VAR robtarget Openhole_4370 := [[433.81, -16, 181.75], [-0.061394, 0.704437, 0.705788, 0.04317], [0,0,0,0], [9E9, 9E9, 9E9, 9E9, 9E9, 9E9]];
	VAR robtarget Openhole_4371 := [[434.8, -16.09, 181.71], [-0.057779, 0.704742, 0.705965, 0.040171], [0,0,0,0], [9E9, 9E9, 9E9, 9E9, 9E9, 9E9]];
	VAR robtarget Openhole_4372 := [[435.3, -16.15, 181.69], [-0.055933, 0.704891, 0.706046, 0.038711], [0,0,0,0], [9E9, 9E9, 9E9, 9E9, 9E9, 9E9]];
	VAR robtarget Openhole_4373 := [[438.22, -12.1, 182.04], [-0.05987, 0.704568, 0.706942, 0.015247], [0,0,0,0], [9E9, 9E9, 9E9, 9E9, 9E9, 9E9]];
	VAR robtarget Openhole_4374 := [[439.21, -12.15, 181.97], [-0.056359, 0.704857, 0.707004, 0.012061], [0,0,0,0], [9E9, 9E9, 9E9, 9E9, 9E9, 9E9]];
	VAR robtarget Openhole_4375 := [[440.21, -12.22, 181.9], [-0.052781, 0.705134, 0.70705, 0.008936], [0,0,0,0], [9E9, 9E9, 9E9, 9E9, 9E9, 9E9]];
	VAR robtarget Openhole_4376 := [[441.7, -12.31, 181.8], [-0.047471, 0.705511, 0.707095, 0.004155], [0,0,0,0], [9E9, 9E9, 9E9, 9E9, 9E9, 9E9]];
	VAR robtarget Openhole_4377 := [[442.2, -12.35, 181.76], [-0.045666, 0.705631, 0.707102, 0.002596], [0,0,0,0], [9E9, 9E9, 9E9, 9E9, 9E9, 9E9]];
	VAR robtarget Openhole_4378 := [[443.19, -12.46, 181.69], [-0.04195, 0.705861, 0.707107, -0.000403], [0,0,0,0], [9E9, 9E9, 9E9, 9E9, 9E9, 9E9]];
	VAR robtarget Openhole_4379 := [[443.92, -12.82, 181.63], [-0.038253, 0.706071, 0.707105, -0.001665], [0,0,0,0], [9E9, 9E9, 9E9, 9E9, 9E9, 9E9]];
	VAR robtarget Openhole_4380 := [[455.86, -14.06, 180.99], [0.006564, 0.707076, 0.706084, -0.038017], [0,0,0,0], [9E9, 9E9, 9E9, 9E9, 9E9, 9E9]];
	VAR robtarget Openhole_4381 := [[456.33, -13.69, 180.94], [0.006897, 0.707073, 0.705926, -0.040852], [0,0,0,0], [9E9, 9E9, 9E9, 9E9, 9E9, 9E9]];
	VAR robtarget Openhole_4382 := [[456.74, -13.4, 180.9], [0.00728, 0.707069, 0.705786, -0.043199], [0,0,0,0], [9E9, 9E9, 9E9, 9E9, 9E9, 9E9]];
	VAR robtarget Openhole_4383 := [[457.15, -13.13, 180.86], [0.007794, 0.707064, 0.70564, -0.045519], [0,0,0,0], [9E9, 9E9, 9E9, 9E9, 9E9, 9E9]];
	VAR robtarget Openhole_4384 := [[457.59, -12.89, 180.81], [0.008483, 0.707056, 0.70549, -0.04779], [0,0,0,0], [9E9, 9E9, 9E9, 9E9, 9E9, 9E9]];
	VAR robtarget Openhole_4385 := [[458.49, -12.46, 180.72], [0.010073, 0.707035, 0.705173, -0.052255], [0,0,0,0], [9E9, 9E9, 9E9, 9E9, 9E9, 9E9]];
	VAR robtarget Openhole_4386 := [[459.4, -12.06, 180.63], [0.011824, 0.707008, 0.704834, -0.056647], [0,0,0,0], [9E9, 9E9, 9E9, 9E9, 9E9, 9E9]];
	VAR robtarget Openhole_4387 := [[461.73, -11.18, 180.37], [0.016707, 0.706909, 0.703892, -0.067348], [0,0,0,0], [9E9, 9E9, 9E9, 9E9, 9E9, 9E9]];
	VAR robtarget Openhole_4388 := [[464.08, -10.39, 180.08], [0.022026, 0.706764, 0.702821, -0.077735], [0,0,0,0], [9E9, 9E9, 9E9, 9E9, 9E9, 9E9]];
	VAR robtarget Openhole_4389 := [[465.51, -9.96, 179.89], [0.025389, 0.706651, 0.702121, -0.08382], [0,0,0,0], [9E9, 9E9, 9E9, 9E9, 9E9, 9E9]];
	VAR robtarget Openhole_4390 := [[468.4, -7.76, 179.23], [0.027798, 0.70656, 0.69994, -0.100422], [0,0,0,0], [9E9, 9E9, 9E9, 9E9, 9E9, 9E9]];
	VAR robtarget Openhole_4391 := [[460.66, -9.48, 180.26], [0.007369, 0.707068, 0.703684, -0.069487], [0,0,0,0], [9E9, 9E9, 9E9, 9E9, 9E9, 9E9]];
	VAR robtarget Openhole_4392 := [[457.75, -10.16, 180.58], [-0.000182, 0.707107, 0.704764, -0.057511], [0,0,0,0], [9E9, 9E9, 9E9, 9E9, 9E9, 9E9]];
	VAR robtarget Openhole_4393 := [[456.79, -10.4, 180.68], [-0.002685, 0.707102, 0.705081, -0.053482], [0,0,0,0], [9E9, 9E9, 9E9, 9E9, 9E9, 9E9]];
	VAR robtarget Openhole_4394 := [[456.31, -10.53, 180.73], [-0.00389, 0.707096, 0.705234, -0.051436], [0,0,0,0], [9E9, 9E9, 9E9, 9E9, 9E9, 9E9]];
	VAR robtarget Openhole_4395 := [[455.82, -10.65, 180.78], [-0.005134, 0.707088, 0.705378, -0.049408], [0,0,0,0], [9E9, 9E9, 9E9, 9E9, 9E9, 9E9]];
	VAR robtarget Openhole_4396 := [[454.86, -10.92, 180.87], [-0.007486, 0.707067, 0.705656, -0.045268], [0,0,0,0], [9E9, 9E9, 9E9, 9E9, 9E9, 9E9]];
	VAR robtarget Openhole_4397 := [[454.39, -11.08, 180.92], [-0.00855, 0.707055, 0.70579, -0.043137], [0,0,0,0], [9E9, 9E9, 9E9, 9E9, 9E9, 9E9]];
	VAR robtarget Openhole_4398 := [[453.93, -11.26, 180.96], [-0.009489, 0.707043, 0.70592, -0.040945], [0,0,0,0], [9E9, 9E9, 9E9, 9E9, 9E9, 9E9]];
	VAR robtarget Openhole_4399 := [[453.3, -11.75, 181.02], [-0.009987, 0.707036, 0.706128, -0.037192], [0,0,0,0], [9E9, 9E9, 9E9, 9E9, 9E9, 9E9]];
	VAR robtarget Openhole_4400 := [[446.72, -11.14, 181.5], [-0.034451, 0.706267, 0.706906, -0.016862], [0,0,0,0], [9E9, 9E9, 9E9, 9E9, 9E9, 9E9]];
	VAR robtarget Openhole_4401 := [[446.16, -10.86, 181.55], [-0.037325, 0.706121, 0.706927, -0.015934], [0,0,0,0], [9E9, 9E9, 9E9, 9E9, 9E9, 9E9]];
	VAR robtarget Openhole_4402 := [[445.18, -10.67, 181.64], [-0.041262, 0.705902, 0.706983, -0.013217], [0,0,0,0], [9E9, 9E9, 9E9, 9E9, 9E9, 9E9]];
	VAR robtarget Openhole_4403 := [[444.69, -10.59, 181.68], [-0.043199, 0.705786, 0.707008, -0.011817], [0,0,0,0], [9E9, 9E9, 9E9, 9E9, 9E9, 9E9]];
	VAR robtarget Openhole_4404 := [[444.19, -10.54, 181.72], [-0.045048, 0.70567, 0.707032, -0.010304], [0,0,0,0], [9E9, 9E9, 9E9, 9E9, 9E9, 9E9]];
	VAR robtarget Openhole_4405 := [[443.69, -10.51, 181.76], [-0.046826, 0.705555, 0.707053, -0.008709], [0,0,0,0], [9E9, 9E9, 9E9, 9E9, 9E9, 9E9]];
	VAR robtarget Openhole_4406 := [[442.7, -10.49, 181.85], [-0.050252, 0.705319, 0.707086, -0.005384], [0,0,0,0], [9E9, 9E9, 9E9, 9E9, 9E9, 9E9]];
	VAR robtarget Openhole_4407 := [[439.21, -10.53, 182.13], [-0.061808, 0.7044, 0.707076, 0.006615], [0,0,0,0], [9E9, 9E9, 9E9, 9E9, 9E9, 9E9]];
	VAR robtarget Openhole_4408 := [[438.71, -10.53, 182.17], [-0.063471, 0.704252, 0.707058, 0.008304], [0,0,0,0], [9E9, 9E9, 9E9, 9E9, 9E9, 9E9]];
	VAR robtarget Openhole_4409 := [[438.21, -10.53, 182.21], [-0.065136, 0.7041, 0.707036, 0.009988], [0,0,0,0], [9E9, 9E9, 9E9, 9E9, 9E9, 9E9]];
	VAR robtarget Openhole_4410 := [[437.72, -10.53, 182.25], [-0.066792, 0.703945, 0.70701, 0.011677], [0,0,0,0], [9E9, 9E9, 9E9, 9E9, 9E9, 9E9]];
	VAR robtarget Openhole_4411 := [[437.22, -10.53, 182.29], [-0.068462, 0.703785, 0.706981, 0.013347], [0,0,0,0], [9E9, 9E9, 9E9, 9E9, 9E9, 9E9]];
	VAR robtarget Openhole_4412 := [[438.63, -8.96, 182.34], [-0.069031, 0.703729, 0.707099, 0.003304], [0,0,0,0], [9E9, 9E9, 9E9, 9E9, 9E9, 9E9]];
	VAR robtarget Openhole_4413 := [[444.58, -8.42, 181.79], [-0.050875, 0.705274, 0.706858, -0.018747], [0,0,0,0], [9E9, 9E9, 9E9, 9E9, 9E9, 9E9]];
	VAR robtarget Openhole_4414 := [[445.07, -8.4, 181.74], [-0.049285, 0.705387, 0.706809, -0.020529], [0,0,0,0], [9E9, 9E9, 9E9, 9E9, 9E9, 9E9]];
	VAR robtarget Openhole_4415 := [[446.57, -8.37, 181.59], [-0.044341, 0.705715, 0.706639, -0.025716], [0,0,0,0], [9E9, 9E9, 9E9, 9E9, 9E9, 9E9]];
	VAR robtarget Openhole_4416 := [[447.06, -8.37, 181.54], [-0.042644, 0.70582, 0.706576, -0.027399], [0,0,0,0], [9E9, 9E9, 9E9, 9E9, 9E9, 9E9]];
	VAR robtarget Openhole_4417 := [[452.53, -8.5, 180.98], [-0.023585, 0.706713, 0.70564, -0.045524], [0,0,0,0], [9E9, 9E9, 9E9, 9E9, 9E9, 9E9]];
	VAR robtarget Openhole_4418 := [[453.03, -8.5, 180.93], [-0.021894, 0.706768, 0.705529, -0.047212], [0,0,0,0], [9E9, 9E9, 9E9, 9E9, 9E9, 9E9]];
	VAR robtarget Openhole_4419 := [[453.53, -8.5, 180.88], [-0.020213, 0.706818, 0.705413, -0.048907], [0,0,0,0], [9E9, 9E9, 9E9, 9E9, 9E9, 9E9]];
	VAR robtarget Openhole_4420 := [[454.03, -8.5, 180.83], [-0.018511, 0.706864, 0.705295, -0.050581], [0,0,0,0], [9E9, 9E9, 9E9, 9E9, 9E9, 9E9]];
	VAR robtarget Openhole_4421 := [[454.52, -8.49, 180.78], [-0.016836, 0.706906, 0.705172, -0.052279], [0,0,0,0], [9E9, 9E9, 9E9, 9E9, 9E9, 9E9]];
	VAR robtarget Openhole_4422 := [[455.02, -8.48, 180.73], [-0.015182, 0.706944, 0.705042, -0.053995], [0,0,0,0], [9E9, 9E9, 9E9, 9E9, 9E9, 9E9]];
	VAR robtarget Openhole_4423 := [[457.01, -8.37, 180.52], [-0.008782, 0.707052, 0.704468, -0.061034], [0,0,0,0], [9E9, 9E9, 9E9, 9E9, 9E9, 9E9]];
	VAR robtarget Openhole_4424 := [[454.64, -6.86, 180.68], [-0.021918, 0.706767, 0.704715, -0.05811], [0,0,0,0], [9E9, 9E9, 9E9, 9E9, 9E9, 9E9]];
	VAR robtarget Openhole_4425 := [[453.65, -6.78, 180.79], [-0.025562, 0.706645, 0.704962, -0.055036], [0,0,0,0], [9E9, 9E9, 9E9, 9E9, 9E9, 9E9]];
	VAR robtarget Openhole_4426 := [[452.66, -6.67, 180.91], [-0.029316, 0.706499, 0.705185, -0.052092], [0,0,0,0], [9E9, 9E9, 9E9, 9E9, 9E9, 9E9]];
	VAR robtarget Openhole_4427 := [[449.69, -6.4, 181.26], [-0.040322, 0.705956, 0.705802, -0.042939], [0,0,0,0], [9E9, 9E9, 9E9, 9E9, 9E9, 9E9]];
	VAR robtarget Openhole_4428 := [[448.2, -6.35, 181.44], [-0.045564, 0.705637, 0.706081, -0.038067], [0,0,0,0], [9E9, 9E9, 9E9, 9E9, 9E9, 9E9]];
	VAR robtarget Openhole_4429 := [[447.71, -6.35, 181.5], [-0.047226, 0.705528, 0.706172, -0.036357], [0,0,0,0], [9E9, 9E9, 9E9, 9E9, 9E9, 9E9]];
	VAR robtarget Openhole_4430 := [[447.21, -6.37, 181.56], [-0.048857, 0.705417, 0.706259, -0.034617], [0,0,0,0], [9E9, 9E9, 9E9, 9E9, 9E9, 9E9]];
	VAR robtarget Openhole_4431 := [[446.22, -6.44, 181.68], [-0.051974, 0.705194, 0.706427, -0.031007], [0,0,0,0], [9E9, 9E9, 9E9, 9E9, 9E9, 9E9]];
	VAR robtarget Openhole_4432 := [[445.24, -6.56, 181.79], [-0.054885, 0.704973, 0.706582, -0.027229], [0,0,0,0], [9E9, 9E9, 9E9, 9E9, 9E9, 9E9]];
	VAR robtarget Openhole_4433 := [[444.74, -6.64, 181.85], [-0.056291, 0.704863, 0.706654, -0.025302], [0,0,0,0], [9E9, 9E9, 9E9, 9E9, 9E9, 9E9]];
	VAR robtarget Openhole_4434 := [[441.88, -4.7, 182.33], [-0.072367, 0.703394, 0.706764, -0.022], [0,0,0,0], [9E9, 9E9, 9E9, 9E9, 9E9, 9E9]];
	VAR robtarget Openhole_4435 := [[439.03, -2.77, 182.92], [-0.088206, 0.701584, 0.70686, -0.018662], [0,0,0,0], [9E9, 9E9, 9E9, 9E9, 9E9, 9E9]];
	VAR robtarget Openhole_4436 := [[445.19, -0.91, 182.03], [-0.073822, 0.703243, 0.705617, -0.045883], [0,0,0,0], [9E9, 9E9, 9E9, 9E9, 9E9, 9E9]];
	VAR robtarget Openhole_4437 := [[446.14, -0.63, 181.87], [-0.071517, 0.703481, 0.705336, -0.050014], [0,0,0,0], [9E9, 9E9, 9E9, 9E9, 9E9, 9E9]];
	VAR robtarget Openhole_4438 := [[447.09, -0.38, 181.71], [-0.069132, 0.703719, 0.705035, -0.054094], [0,0,0,0], [9E9, 9E9, 9E9, 9E9, 9E9, 9E9]];
	VAR robtarget Openhole_4439 := [[447.57, -0.24, 181.62], [-0.067981, 0.703831, 0.704873, -0.056155], [0,0,0,0], [9E9, 9E9, 9E9, 9E9, 9E9, 9E9]];
	VAR robtarget Openhole_4440 := [[448.05, -0.13, 181.54], [-0.066749, 0.703949, 0.70471, -0.058167], [0,0,0,0], [9E9, 9E9, 9E9, 9E9, 9E9, 9E9]];
	VAR robtarget Openhole_4441 := [[448.52, 0, 181.45], [-0.065551, 0.704062, 0.70454, -0.060198], [0,0,0,0], [9E9, 9E9, 9E9, 9E9, 9E9, 9E9]];
	VAR robtarget Openhole_4442 := [[449.49, 0.16, 181.27], [-0.062782, 0.704314, 0.704203, -0.064017], [0,0,0,0], [9E9, 9E9, 9E9, 9E9, 9E9, 9E9]];
	VAR robtarget Openhole_4443 := [[450.48, 0.12, 181.09], [-0.059329, 0.704613, 0.703903, -0.06723], [0,0,0,0], [9E9, 9E9, 9E9, 9E9, 9E9, 9E9]];
	VAR robtarget Openhole_4444 := [[451.43, -0.1, 180.92], [-0.055316, 0.70494, 0.703662, -0.069716], [0,0,0,0], [9E9, 9E9, 9E9, 9E9, 9E9, 9E9]];
	VAR robtarget Openhole_4445 := [[451.9, -0.27, 180.84], [-0.053183, 0.705104, 0.703561, -0.070729], [0,0,0,0], [9E9, 9E9, 9E9, 9E9, 9E9, 9E9]];
	VAR robtarget Openhole_4446 := [[452.84, -0.58, 180.68], [-0.048971, 0.705409, 0.703341, -0.07288], [0,0,0,0], [9E9, 9E9, 9E9, 9E9, 9E9, 9E9]];
	VAR robtarget Openhole_4447 := [[453.8, -0.8, 180.52], [-0.044957, 0.705676, 0.703077, -0.075384], [0,0,0,0], [9E9, 9E9, 9E9, 9E9, 9E9, 9E9]];
	VAR robtarget Openhole_4448 := [[454.77, -0.99, 180.36], [-0.041014, 0.705916, 0.702792, -0.077996], [0,0,0,0], [9E9, 9E9, 9E9, 9E9, 9E9, 9E9]];
	VAR robtarget Openhole_4449 := [[457.2, -1.38, 179.97], [-0.031405, 0.706409, 0.701996, -0.084866], [0,0,0,0], [9E9, 9E9, 9E9, 9E9, 9E9, 9E9]];
	VAR robtarget Openhole_4450 := [[459.17, -1.56, 179.65], [-0.024076, 0.706697, 0.701256, -0.090777], [0,0,0,0], [9E9, 9E9, 9E9, 9E9, 9E9, 9E9]];
	VAR robtarget Openhole_4451 := [[460.16, -1.6, 179.49], [-0.020553, 0.706808, 0.700848, -0.093873], [0,0,0,0], [9E9, 9E9, 9E9, 9E9, 9E9, 9E9]];
	VAR robtarget Openhole_4452 := [[461.14, -1.61, 179.32], [-0.017136, 0.706899, 0.700413, -0.097063], [0,0,0,0], [9E9, 9E9, 9E9, 9E9, 9E9, 9E9]];
	VAR robtarget Openhole_4453 := [[461.64, -1.61, 179.24], [-0.015457, 0.706938, 0.700187, -0.09868], [0,0,0,0], [9E9, 9E9, 9E9, 9E9, 9E9, 9E9]];
	VAR robtarget Openhole_4454 := [[467.04, -1.32, 178.28], [0.002033, 0.707104, 0.697355, -0.117029], [0,0,0,0], [9E9, 9E9, 9E9, 9E9, 9E9, 9E9]];
	VAR robtarget Openhole_4455 := [[474.41, -0.89, 176.93], [0.025454, 0.706648, 0.692853, -0.14126], [0,0,0,0], [9E9, 9E9, 9E9, 9E9, 9E9, 9E9]];
	VAR robtarget Openhole_4456 := [[476.87, -0.86, 176.49], [0.033531, 0.706311, 0.691282, -0.148758], [0,0,0,0], [9E9, 9E9, 9E9, 9E9, 9E9, 9E9]];
	VAR robtarget Openhole_4457 := [[477.36, -0.86, 176.4], [0.035168, 0.706232, 0.690967, -0.150215], [0,0,0,0], [9E9, 9E9, 9E9, 9E9, 9E9, 9E9]];
	VAR robtarget Openhole_4458 := [[482.78, -1.08, 175.52], [0.05357, 0.705075, 0.687507, -0.165332], [0,0,0,0], [9E9, 9E9, 9E9, 9E9, 9E9, 9E9]];
	VAR robtarget Openhole_4459 := [[488.7, -1.64, 174.71], [0.07413, 0.70321, 0.683789, -0.180092], [0,0,0,0], [9E9, 9E9, 9E9, 9E9, 9E9, 9E9]];
	VAR robtarget Openhole_4460 := [[495.1, -2.58, 174.06], [0.096562, 0.700483, 0.679902, -0.194249], [0,0,0,0], [9E9, 9E9, 9E9, 9E9, 9E9, 9E9]];
	VAR robtarget Openhole_4461 := [[495.59, -2.66, 174.01], [0.098281, 0.700243, 0.679611, -0.195267], [0,0,0,0], [9E9, 9E9, 9E9, 9E9, 9E9, 9E9]];
	VAR robtarget Openhole_4462 := [[495.54, -3.95, 174.59], [0.101997, 0.699712, 0.68072, -0.191363], [0,0,0,0], [9E9, 9E9, 9E9, 9E9, 9E9, 9E9]];
	VAR robtarget Openhole_4463 := [[488.63, -3.04, 175.25], [0.078211, 0.702768, 0.68493, -0.1757], [0,0,0,0], [9E9, 9E9, 9E9, 9E9, 9E9, 9E9]];
	VAR robtarget Openhole_4464 := [[482.7, -2.51, 176], [0.057814, 0.704739, 0.688609, -0.160678], [0,0,0,0], [9E9, 9E9, 9E9, 9E9, 9E9, 9E9]];
	VAR robtarget Openhole_4465 := [[477.26, -2.32, 176.81], [0.039496, 0.706003, 0.692001, -0.145378], [0,0,0,0], [9E9, 9E9, 9E9, 9E9, 9E9, 9E9]];
	VAR robtarget Openhole_4466 := [[476.77, -2.31, 176.89], [0.037862, 0.706092, 0.692308, -0.143908], [0,0,0,0], [9E9, 9E9, 9E9, 9E9, 9E9, 9E9]];
	VAR robtarget Openhole_4467 := [[476.28, -2.32, 176.97], [0.036243, 0.706177, 0.692616, -0.142417], [0,0,0,0], [9E9, 9E9, 9E9, 9E9, 9E9, 9E9]];
	VAR robtarget Openhole_4468 := [[470.37, -2.56, 177.97], [0.017293, 0.706895, 0.696233, -0.123531], [0,0,0,0], [9E9, 9E9, 9E9, 9E9, 9E9, 9E9]];
	VAR robtarget Openhole_4469 := [[462.5, -3.12, 179.29], [-0.00753, 0.707067, 0.700484, -0.096549], [0,0,0,0], [9E9, 9E9, 9E9, 9E9, 9E9, 9E9]];
	VAR robtarget Openhole_4470 := [[461.51, -3.15, 179.44], [-0.010802, 0.707024, 0.700934, -0.093227], [0,0,0,0], [9E9, 9E9, 9E9, 9E9, 9E9, 9E9]];
	VAR robtarget Openhole_4471 := [[461.02, -3.16, 179.52], [-0.012484, 0.706997, 0.701148, -0.091602], [0,0,0,0], [9E9, 9E9, 9E9, 9E9, 9E9, 9E9]];
	VAR robtarget Openhole_4472 := [[460.52, -3.16, 179.59], [-0.014175, 0.706965, 0.701358, -0.089981], [0,0,0,0], [9E9, 9E9, 9E9, 9E9, 9E9, 9E9]];
	VAR robtarget Openhole_4473 := [[459.53, -3.13, 179.74], [-0.01764, 0.706887, 0.701758, -0.086812], [0,0,0,0], [9E9, 9E9, 9E9, 9E9, 9E9, 9E9]];
	VAR robtarget Openhole_4474 := [[458.54, -3.07, 179.89], [-0.021205, 0.706789, 0.702131, -0.083734], [0,0,0,0], [9E9, 9E9, 9E9, 9E9, 9E9, 9E9]];
	VAR robtarget Openhole_4475 := [[454.62, -2.55, 180.46], [-0.036367, 0.706171, 0.703389, -0.072411], [0,0,0,0], [9E9, 9E9, 9E9, 9E9, 9E9, 9E9]];
	VAR robtarget Openhole_4476 := [[451.22, -1.9, 180.99], [-0.0501, 0.70533, 0.704286, -0.063093], [0,0,0,0], [9E9, 9E9, 9E9, 9E9, 9E9, 9E9]];
	VAR robtarget Openhole_4477 := [[450.73, -1.83, 181.07], [-0.051992, 0.705193, 0.704413, -0.061667], [0,0,0,0], [9E9, 9E9, 9E9, 9E9, 9E9, 9E9]];
	VAR robtarget Openhole_4478 := [[450.24, -1.78, 181.15], [-0.053831, 0.705055, 0.704542, -0.060176], [0,0,0,0], [9E9, 9E9, 9E9, 9E9, 9E9, 9E9]];
	VAR robtarget Openhole_4479 := [[449.75, -1.74, 181.23], [-0.055631, 0.704915, 0.704671, -0.058637], [0,0,0,0], [9E9, 9E9, 9E9, 9E9, 9E9, 9E9]];
	VAR robtarget Openhole_4480 := [[449.26, -1.74, 181.32], [-0.057315, 0.70478, 0.704808, -0.056975], [0,0,0,0], [9E9, 9E9, 9E9, 9E9, 9E9, 9E9]];
	VAR robtarget Openhole_4481 := [[448.77, -1.75, 181.4], [-0.058951, 0.704645, 0.704944, -0.055262], [0,0,0,0], [9E9, 9E9, 9E9, 9E9, 9E9, 9E9]];
	VAR robtarget Openhole_4482 := [[448.27, -1.79, 181.48], [-0.0605, 0.704514, 0.705082, -0.053471], [0,0,0,0], [9E9, 9E9, 9E9, 9E9, 9E9, 9E9]];
	VAR robtarget Openhole_4483 := [[447.78, -1.85, 181.56], [-0.061951, 0.704388, 0.705221, -0.051602], [0,0,0,0], [9E9, 9E9, 9E9, 9E9, 9E9, 9E9]];
	VAR robtarget Openhole_4484 := [[447.3, -1.93, 181.64], [-0.063351, 0.704263, 0.705359, -0.04969], [0,0,0,0], [9E9, 9E9, 9E9, 9E9, 9E9, 9E9]];
	VAR robtarget Openhole_4485 := [[446.81, -2.01, 181.72], [-0.064707, 0.70414, 0.705493, -0.047749], [0,0,0,0], [9E9, 9E9, 9E9, 9E9, 9E9, 9E9]];
	VAR robtarget Openhole_4486 := [[445.84, -2.22, 181.87], [-0.067271, 0.7039, 0.705751, -0.043762], [0,0,0,0], [9E9, 9E9, 9E9, 9E9, 9E9, 9E9]];
	VAR robtarget Openhole_4487 := [[444.89, -2.47, 182.01], [-0.069682, 0.703665, 0.705993, -0.039677], [0,0,0,0], [9E9, 9E9, 9E9, 9E9, 9E9, 9E9]];
	VAR robtarget Openhole_4488 := [[438.19, -4.32, 182.88], [-0.085872, 0.701873, 0.707026, -0.010686], [0,0,0,0], [9E9, 9E9, 9E9, 9E9, 9E9, 9E9]];
	VAR robtarget Openhole_4489 := [[437.22, -4.54, 182.99], [-0.088344, 0.701566, 0.707075, -0.006658], [0,0,0,0], [9E9, 9E9, 9E9, 9E9, 9E9, 9E9]];
	VAR robtarget Openhole_4490 := [[431.68, -6.99, 183.35], [-0.098305, 0.70024, 0.706816, 0.020274], [0,0,0,0], [9E9, 9E9, 9E9, 9E9, 9E9, 9E9]];
	VAR robtarget Openhole_4491 := [[438.07, -6.03, 182.71], [-0.08061, 0.702497, 0.707092, -0.004586], [0,0,0,0], [9E9, 9E9, 9E9, 9E9, 9E9, 9E9]];
	VAR robtarget Openhole_4492 := [[444.39, -4.68, 181.99], [-0.064023, 0.704202, 0.706443, -0.030626], [0,0,0,0], [9E9, 9E9, 9E9, 9E9, 9E9, 9E9]];
	VAR robtarget Openhole_4493 := [[444.87, -4.57, 181.92], [-0.062758, 0.704316, 0.706353, -0.032641], [0,0,0,0], [9E9, 9E9, 9E9, 9E9, 9E9, 9E9]];
	VAR robtarget Openhole_4494 := [[445.84, -4.38, 181.8], [-0.060138, 0.704545, 0.706158, -0.036613], [0,0,0,0], [9E9, 9E9, 9E9, 9E9, 9E9, 9E9]];
	VAR robtarget Openhole_4495 := [[446.33, -4.29, 181.73], [-0.058773, 0.70466, 0.706055, -0.03856], [0,0,0,0], [9E9, 9E9, 9E9, 9E9, 9E9, 9E9]];
	VAR robtarget Openhole_4496 := [[446.82, -4.21, 181.66], [-0.057372, 0.704775, 0.705947, -0.040482], [0,0,0,0], [9E9, 9E9, 9E9, 9E9, 9E9, 9E9]];
	VAR robtarget Openhole_4497 := [[447.31, -4.15, 181.59], [-0.055926, 0.704892, 0.705836, -0.042369], [0,0,0,0], [9E9, 9E9, 9E9, 9E9, 9E9, 9E9]];
	VAR robtarget Openhole_4498 := [[447.8, -4.1, 181.52], [-0.054421, 0.705009, 0.705723, -0.04421], [0,0,0,0], [9E9, 9E9, 9E9, 9E9, 9E9, 9E9]];
	VAR robtarget Openhole_4499 := [[448.3, -4.06, 181.45], [-0.052883, 0.705127, 0.705608, -0.046022], [0,0,0,0], [9E9, 9E9, 9E9, 9E9, 9E9, 9E9]];
	VAR robtarget Openhole_4500 := [[448.79, -4.06, 181.38], [-0.051205, 0.70525, 0.705496, -0.047705], [0,0,0,0], [9E9, 9E9, 9E9, 9E9, 9E9, 9E9]];
	VAR robtarget Openhole_4501 := [[449.78, -4.1, 181.24], [-0.047721, 0.705495, 0.70527, -0.05094], [0,0,0,0], [9E9, 9E9, 9E9, 9E9, 9E9, 9E9]];
	VAR robtarget Openhole_4502 := [[450.77, -4.2, 181.1], [-0.044031, 0.705735, 0.705046, -0.05394], [0,0,0,0], [9E9, 9E9, 9E9, 9E9, 9E9, 9E9]];
	VAR robtarget Openhole_4503 := [[456.16, -5.01, 180.38], [-0.022926, 0.706735, 0.703693, -0.0694], [0,0,0,0], [9E9, 9E9, 9E9, 9E9, 9E9, 9E9]];
	VAR robtarget Openhole_4504 := [[458.63, -5.19, 180.06], [-0.013857, 0.706971, 0.7029, -0.077018], [0,0,0,0], [9E9, 9E9, 9E9, 9E9, 9E9, 9E9]];
	VAR robtarget Openhole_4505 := [[459.13, -5.2, 180], [-0.012129, 0.707003, 0.702722, -0.078627], [0,0,0,0], [9E9, 9E9, 9E9, 9E9, 9E9, 9E9]];
	VAR robtarget Openhole_4506 := [[463.08, -5.04, 179.45], [0.00081, 0.707106, 0.701072, -0.092185], [0,0,0,0], [9E9, 9E9, 9E9, 9E9, 9E9, 9E9]];
	VAR robtarget Openhole_4507 := [[464.07, -4.96, 179.31], [0.003891, 0.707096, 0.700606, -0.095663], [0,0,0,0], [9E9, 9E9, 9E9, 9E9, 9E9, 9E9]];
	VAR robtarget Openhole_4508 := [[472.91, -4.06, 177.9], [0.030712, 0.706439, 0.695675, -0.126635], [0,0,0,0], [9E9, 9E9, 9E9, 9E9, 9E9, 9E9]];
	VAR robtarget Openhole_4509 := [[478.34, -3.86, 177.07], [0.04798, 0.705477, 0.692339, -0.143757], [0,0,0,0], [9E9, 9E9, 9E9, 9E9, 9E9, 9E9]];
	VAR robtarget Openhole_4510 := [[478.84, -3.85, 176.99], [0.04959, 0.705366, 0.692032, -0.145232], [0,0,0,0], [9E9, 9E9, 9E9, 9E9, 9E9, 9E9]];
	VAR robtarget Openhole_4511 := [[479.33, -3.86, 176.92], [0.051212, 0.70525, 0.691725, -0.146687], [0,0,0,0], [9E9, 9E9, 9E9, 9E9, 9E9, 9E9]];
	VAR robtarget Openhole_4512 := [[480.82, -3.88, 176.71], [0.056107, 0.704877, 0.690802, -0.150974], [0,0,0,0], [9E9, 9E9, 9E9, 9E9, 9E9, 9E9]];
	VAR robtarget Openhole_4513 := [[474.12, -5.49, 178.07], [0.039383, 0.706009, 0.695836, -0.125746], [0,0,0,0], [9E9, 9E9, 9E9, 9E9, 9E9, 9E9]];
	VAR robtarget Openhole_4514 := [[469.2, -6.03, 178.82], [0.024778, 0.706673, 0.698712, -0.108635], [0,0,0,0], [9E9, 9E9, 9E9, 9E9, 9E9, 9E9]];
	VAR robtarget Openhole_4515 := [[460.88, -7.27, 180], [0.00075, 0.707106, 0.70284, -0.077563], [0,0,0,0], [9E9, 9E9, 9E9, 9E9, 9E9, 9E9]];
	VAR robtarget Openhole_4516 := [[457.42, -7.57, 180.41], [-0.010066, 0.707035, 0.704105, -0.065081], [0,0,0,0], [9E9, 9E9, 9E9, 9E9, 9E9, 9E9]];
	VAR robtarget Openhole_4517 := [[455.43, -7.61, 180.63], [-0.016702, 0.706909, 0.704701, -0.05828], [0,0,0,0], [9E9, 9E9, 9E9, 9E9, 9E9, 9E9]];
	VAR robtarget Openhole_4518 := [[452.45, -7.48, 180.96], [-0.027313, 0.706579, 0.705429, -0.048681], [0,0,0,0], [9E9, 9E9, 9E9, 9E9, 9E9, 9E9]];
	VAR robtarget Openhole_4519 := [[448.48, -7.26, 181.4], [-0.041571, 0.705884, 0.706192, -0.035963], [0,0,0,0], [9E9, 9E9, 9E9, 9E9, 9E9, 9E9]];
	VAR robtarget Openhole_4520 := [[447.49, -7.25, 181.51], [-0.044979, 0.705675, 0.706354, -0.032618], [0,0,0,0], [9E9, 9E9, 9E9, 9E9, 9E9, 9E9]];
	VAR robtarget Openhole_4521 := [[446.49, -7.27, 181.62], [-0.04828, 0.705457, 0.706505, -0.029169], [0,0,0,0], [9E9, 9E9, 9E9, 9E9, 9E9, 9E9]];
	VAR robtarget Openhole_4522 := [[445.5, -7.33, 181.73], [-0.05141, 0.705235, 0.706644, -0.025565], [0,0,0,0], [9E9, 9E9, 9E9, 9E9, 9E9, 9E9]];
	VAR robtarget Openhole_4523 := [[444.51, -7.43, 181.84], [-0.054417, 0.70501, 0.706769, -0.02186], [0,0,0,0], [9E9, 9E9, 9E9, 9E9, 9E9, 9E9]];
	VAR robtarget Openhole_4524 := [[444.02, -7.49, 181.89], [-0.055888, 0.704895, 0.706824, -0.019981], [0,0,0,0], [9E9, 9E9, 9E9, 9E9, 9E9, 9E9]];
	VAR robtarget Openhole_4525 := [[437.6, -8.31, 182.51], [-0.074579, 0.703163, 0.707092, 0.004624], [0,0,0,0], [9E9, 9E9, 9E9, 9E9, 9E9, 9E9]];
	VAR robtarget Openhole_4526 := [[423.69, -9.33, 183.7], [-0.115934, 0.697538, 0.705007, 0.054452], [0,0,0,0], [9E9, 9E9, 9E9, 9E9, 9E9, 9E9]];
	VAR robtarget Openhole_4527 := [[407.25, -10.08, 184.93], [-0.161886, 0.688326, 0.698774, 0.108234], [0,0,0,0], [9E9, 9E9, 9E9, 9E9, 9E9, 9E9]];
	VAR robtarget Openhole_4528 := [[394.36, -10.64, 185.74], [-0.19397, 0.679982, 0.691771, 0.146468], [0,0,0,0], [9E9, 9E9, 9E9, 9E9, 9E9, 9E9]];
	VAR robtarget Openhole_4529 := [[389.36, -10.64, 186.14], [-0.206026, 0.676427, 0.688852, 0.159635], [0,0,0,0], [9E9, 9E9, 9E9, 9E9, 9E9, 9E9]];
	VAR robtarget Openhole_4530 := [[362.36, -10.64, 186.23], [-0.183051, 0.683002, 0.683002, 0.183051], [0,0,0,0], [9E9, 9E9, 9E9, 9E9, 9E9, 9E9]];
	VAR robtarget Openhole_4531 := [[361.72, -33.92, 172.78], [-0.183051, 0.683002, 0.683002, 0.183051], [0,0,0,0], [9E9, 9E9, 9E9, 9E9, 9E9, 9E9]];
	VAR robtarget Openhole_4532 := [[389.32, -33.92, 172.7], [-0.139779, 0.693153, 0.670225, 0.225385], [0,0,0,0], [9E9, 9E9, 9E9, 9E9, 9E9, 9E9]];
	VAR robtarget Openhole_4533 := [[399.12, -33.92, 174.1], [-0.112383, 0.698119, 0.677552, 0.202294], [0,0,0,0], [9E9, 9E9, 9E9, 9E9, 9E9, 9E9]];
	VAR robtarget Openhole_4534 := [[405.5, -35.06, 174.54], [-0.089977, 0.701359, 0.681274, 0.189382], [0,0,0,0], [9E9, 9E9, 9E9, 9E9, 9E9, 9E9]];
	VAR robtarget Openhole_4535 := [[411.91, -35.92, 175.22], [-0.067429, 0.703884, 0.685171, 0.174758], [0,0,0,0], [9E9, 9E9, 9E9, 9E9, 9E9, 9E9]];
	VAR robtarget Openhole_4536 := [[417.84, -36.39, 176.04], [-0.046877, 0.705551, 0.688882, 0.159505], [0,0,0,0], [9E9, 9E9, 9E9, 9E9, 9E9, 9E9]];
	VAR robtarget Openhole_4537 := [[421.78, -36.5, 176.67], [-0.033524, 0.706312, 0.691381, 0.148297], [0,0,0,0], [9E9, 9E9, 9E9, 9E9, 9E9, 9E9]];
	VAR robtarget Openhole_4538 := [[422.28, -36.5, 176.75], [-0.031888, 0.706387, 0.691694, 0.146829], [0,0,0,0], [9E9, 9E9, 9E9, 9E9, 9E9, 9E9]];
	VAR robtarget Openhole_4539 := [[428.18, -36.31, 177.78], [-0.012722, 0.706992, 0.695381, 0.128239], [0,0,0,0], [9E9, 9E9, 9E9, 9E9, 9E9, 9E9]];
	VAR robtarget Openhole_4540 := [[436.05, -35.81, 179.15], [0.012415, 0.706998, 0.699758, 0.101677], [0,0,0,0], [9E9, 9E9, 9E9, 9E9, 9E9, 9E9]];
	VAR robtarget Openhole_4541 := [[437.03, -35.79, 179.32], [0.01572, 0.706932, 0.700226, 0.098405], [0,0,0,0], [9E9, 9E9, 9E9, 9E9, 9E9, 9E9]];
	VAR robtarget Openhole_4542 := [[438.02, -35.8, 179.47], [0.019111, 0.706848, 0.70067, 0.095196], [0,0,0,0], [9E9, 9E9, 9E9, 9E9, 9E9, 9E9]];
	VAR robtarget Openhole_4543 := [[439.01, -35.82, 179.63], [0.022586, 0.706746, 0.701089, 0.092055], [0,0,0,0], [9E9, 9E9, 9E9, 9E9, 9E9, 9E9]];
	VAR robtarget Openhole_4544 := [[440, -35.88, 179.79], [0.02616, 0.706623, 0.701483, 0.089007], [0,0,0,0], [9E9, 9E9, 9E9, 9E9, 9E9, 9E9]];
	VAR robtarget Openhole_4545 := [[440.98, -35.98, 179.94], [0.02983, 0.706477, 0.701851, 0.086055], [0,0,0,0], [9E9, 9E9, 9E9, 9E9, 9E9, 9E9]];
	VAR robtarget Openhole_4546 := [[441.96, -36.1, 180.09], [0.033602, 0.706308, 0.702193, 0.083218], [0,0,0,0], [9E9, 9E9, 9E9, 9E9, 9E9, 9E9]];
	VAR robtarget Openhole_4547 := [[442.94, -36.26, 180.24], [0.037457, 0.706114, 0.702511, 0.080485], [0,0,0,0], [9E9, 9E9, 9E9, 9E9, 9E9, 9E9]];
	VAR robtarget Openhole_4548 := [[443.91, -36.44, 180.39], [0.041385, 0.705895, 0.702808, 0.077851], [0,0,0,0], [9E9, 9E9, 9E9, 9E9, 9E9, 9E9]];
	VAR robtarget Openhole_4549 := [[445.84, -36.87, 180.7], [0.049371, 0.705381, 0.703352, 0.072777], [0,0,0,0], [9E9, 9E9, 9E9, 9E9, 9E9, 9E9]];
	VAR robtarget Openhole_4550 := [[446.31, -37, 180.78], [0.051445, 0.705233, 0.703468, 0.071641], [0,0,0,0], [9E9, 9E9, 9E9, 9E9, 9E9, 9E9]];
	VAR robtarget Openhole_4551 := [[446.78, -37.17, 180.85], [0.053574, 0.705074, 0.703572, 0.070614], [0,0,0,0], [9E9, 9E9, 9E9, 9E9, 9E9, 9E9]];
	VAR robtarget Openhole_4552 := [[447.24, -37.35, 180.93], [0.055739, 0.704907, 0.703666, 0.069672], [0,0,0,0], [9E9, 9E9, 9E9, 9E9, 9E9, 9E9]];
	VAR robtarget Openhole_4553 := [[448.2, -37.57, 181.1], [0.059719, 0.70458, 0.703913, 0.067134], [0,0,0,0], [9E9, 9E9, 9E9, 9E9, 9E9, 9E9]];
	VAR robtarget Openhole_4554 := [[448.69, -37.57, 181.18], [0.061409, 0.704435, 0.704067, 0.06549], [0,0,0,0], [9E9, 9E9, 9E9, 9E9, 9E9, 9E9]];
	VAR robtarget Openhole_4555 := [[449.18, -37.57, 181.27], [0.063054, 0.70429, 0.704223, 0.063801], [0,0,0,0], [9E9, 9E9, 9E9, 9E9, 9E9, 9E9]];
	VAR robtarget Openhole_4556 := [[450.15, -37.36, 181.44], [0.065651, 0.704052, 0.704568, 0.059864], [0,0,0,0], [9E9, 9E9, 9E9, 9E9, 9E9, 9E9]];
	VAR robtarget Openhole_4557 := [[450.62, -37.23, 181.52], [0.066831, 0.703941, 0.704739, 0.057822], [0,0,0,0], [9E9, 9E9, 9E9, 9E9, 9E9, 9E9]];
	VAR robtarget Openhole_4558 := [[451.1, -37.12, 181.61], [0.068071, 0.703823, 0.704901, 0.055814], [0,0,0,0], [9E9, 9E9, 9E9, 9E9, 9E9, 9E9]];
	VAR robtarget Openhole_4559 := [[451.58, -36.98, 181.69], [0.069229, 0.70371, 0.705061, 0.053756], [0,0,0,0], [9E9, 9E9, 9E9, 9E9, 9E9, 9E9]];
	VAR robtarget Openhole_4560 := [[459.65, -34.59, 182.84], [0.088256, 0.701577, 0.70687, 0.018282], [0,0,0,0], [9E9, 9E9, 9E9, 9E9, 9E9, 9E9]];
	VAR robtarget Openhole_4561 := [[460.13, -34.45, 182.9], [0.089394, 0.701433, 0.706921, 0.016207], [0,0,0,0], [9E9, 9E9, 9E9, 9E9, 9E9, 9E9]];
	VAR robtarget Openhole_4562 := [[461.11, -32.96, 182.88], [0.087702, 0.701647, 0.707063, 0.007906], [0,0,0,0], [9E9, 9E9, 9E9, 9E9, 9E9, 9E9]];
	VAR robtarget Openhole_4563 := [[460.14, -33.18, 182.77], [0.085245, 0.70195, 0.707006, 0.011948], [0,0,0,0], [9E9, 9E9, 9E9, 9E9, 9E9, 9E9]];
	VAR robtarget Openhole_4564 := [[453.43, -34.99, 181.93], [0.068918, 0.70374, 0.705924, 0.040876], [0,0,0,0], [9E9, 9E9, 9E9, 9E9, 9E9, 9E9]];
	VAR robtarget Openhole_4565 := [[452.47, -35.23, 181.79], [0.066442, 0.703978, 0.705678, 0.044922], [0,0,0,0], [9E9, 9E9, 9E9, 9E9, 9E9, 9E9]];
	VAR robtarget Openhole_4566 := [[451.98, -35.33, 181.72], [0.065155, 0.704099, 0.705549, 0.046912], [0,0,0,0], [9E9, 9E9, 9E9, 9E9, 9E9, 9E9]];
	VAR robtarget Openhole_4567 := [[451.5, -35.42, 181.64], [0.063827, 0.70422, 0.705416, 0.048874], [0,0,0,0], [9E9, 9E9, 9E9, 9E9, 9E9, 9E9]];
	VAR robtarget Openhole_4568 := [[451.01, -35.49, 181.56], [0.062401, 0.704348, 0.705282, 0.050766], [0,0,0,0], [9E9, 9E9, 9E9, 9E9, 9E9, 9E9]];
	VAR robtarget Openhole_4569 := [[450.52, -35.55, 181.49], [0.060929, 0.704477, 0.705146, 0.05262], [0,0,0,0], [9E9, 9E9, 9E9, 9E9, 9E9, 9E9]];
	VAR robtarget Openhole_4570 := [[450.03, -35.58, 181.41], [0.059378, 0.704609, 0.70501, 0.054409], [0,0,0,0], [9E9, 9E9, 9E9, 9E9, 9E9, 9E9]];
	VAR robtarget Openhole_4571 := [[449.53, -35.6, 181.33], [0.057764, 0.704743, 0.704874, 0.056143], [0,0,0,0], [9E9, 9E9, 9E9, 9E9, 9E9, 9E9]];
	VAR robtarget Openhole_4572 := [[449.04, -35.59, 181.25], [0.056048, 0.704882, 0.704743, 0.057773], [0,0,0,0], [9E9, 9E9, 9E9, 9E9, 9E9, 9E9]];
	VAR robtarget Openhole_4573 := [[448.55, -35.55, 181.17], [0.054253, 0.705022, 0.704614, 0.059318], [0,0,0,0], [9E9, 9E9, 9E9, 9E9, 9E9, 9E9]];
	VAR robtarget Openhole_4574 := [[448.06, -35.5, 181.1], [0.052405, 0.705162, 0.704488, 0.060799], [0,0,0,0], [9E9, 9E9, 9E9, 9E9, 9E9, 9E9]];
	VAR robtarget Openhole_4575 := [[447.57, -35.43, 181.02], [0.050507, 0.705301, 0.704364, 0.062216], [0,0,0,0], [9E9, 9E9, 9E9, 9E9, 9E9, 9E9]];
	VAR robtarget Openhole_4576 := [[446.59, -35.25, 180.87], [0.0466, 0.70557, 0.704122, 0.0649], [0,0,0,0], [9E9, 9E9, 9E9, 9E9, 9E9, 9E9]];
	VAR robtarget Openhole_4577 := [[443.68, -34.65, 180.45], [0.034704, 0.706255, 0.703358, 0.072716], [0,0,0,0], [9E9, 9E9, 9E9, 9E9, 9E9, 9E9]];
	VAR robtarget Openhole_4578 := [[441.73, -34.35, 180.18], [0.02701, 0.706591, 0.702764, 0.078249], [0,0,0,0], [9E9, 9E9, 9E9, 9E9, 9E9, 9E9]];
	VAR robtarget Openhole_4579 := [[440.74, -34.25, 180.04], [0.023295, 0.706723, 0.702432, 0.081175], [0,0,0,0], [9E9, 9E9, 9E9, 9E9, 9E9, 9E9]];
	VAR robtarget Openhole_4580 := [[439.75, -34.17, 179.9], [0.019671, 0.706833, 0.702076, 0.084198], [0,0,0,0], [9E9, 9E9, 9E9, 9E9, 9E9, 9E9]];
	VAR robtarget Openhole_4581 := [[438.76, -34.13, 179.76], [0.016144, 0.706922, 0.701695, 0.087315], [0,0,0,0], [9E9, 9E9, 9E9, 9E9, 9E9, 9E9]];
	VAR robtarget Openhole_4582 := [[437.77, -34.12, 179.62], [0.012723, 0.706992, 0.701288, 0.090526], [0,0,0,0], [9E9, 9E9, 9E9, 9E9, 9E9, 9E9]];
	VAR robtarget Openhole_4583 := [[437.28, -34.12, 179.55], [0.011048, 0.70702, 0.701075, 0.092159], [0,0,0,0], [9E9, 9E9, 9E9, 9E9, 9E9, 9E9]];
	VAR robtarget Openhole_4584 := [[431.85, -34.44, 178.71], [-0.006374, 0.707078, 0.698386, 0.11071], [0,0,0,0], [9E9, 9E9, 9E9, 9E9, 9E9, 9E9]];
	VAR robtarget Openhole_4585 := [[424.96, -34.89, 177.58], [-0.028142, 0.706547, 0.694362, 0.133646], [0,0,0,0], [9E9, 9E9, 9E9, 9E9, 9E9, 9E9]];
	VAR robtarget Openhole_4586 := [[422, -34.94, 177.11], [-0.037815, 0.706095, 0.692544, 0.142768], [0,0,0,0], [9E9, 9E9, 9E9, 9E9, 9E9, 9E9]];
	VAR robtarget Openhole_4587 := [[421.5, -34.94, 177.04], [-0.039458, 0.706005, 0.692241, 0.144233], [0,0,0,0], [9E9, 9E9, 9E9, 9E9, 9E9, 9E9]];
	VAR robtarget Openhole_4588 := [[415.57, -34.71, 176.21], [-0.059556, 0.704594, 0.688577, 0.160815], [0,0,0,0], [9E9, 9E9, 9E9, 9E9, 9E9, 9E9]];
	VAR robtarget Openhole_4589 := [[409.14, -34.09, 175.47], [-0.081789, 0.702361, 0.684641, 0.176824], [0,0,0,0], [9E9, 9E9, 9E9, 9E9, 9E9, 9E9]];
	VAR robtarget Openhole_4590 := [[404.2, -33.45, 175.04], [-0.098838, 0.700165, 0.681654, 0.18801], [0,0,0,0], [9E9, 9E9, 9E9, 9E9, 9E9, 9E9]];
	VAR robtarget Openhole_4591 := [[411.67, -32.92, 176.27], [-0.077558, 0.70284, 0.687273, 0.1663], [0,0,0,0], [9E9, 9E9, 9E9, 9E9, 9E9, 9E9]];
	VAR robtarget Openhole_4592 := [[418.12, -33.28, 177.02], [-0.055864, 0.704897, 0.691226, 0.149019], [0,0,0,0], [9E9, 9E9, 9E9, 9E9, 9E9, 9E9]];
	VAR robtarget Openhole_4593 := [[420.59, -33.32, 177.35], [-0.047674, 0.705498, 0.692738, 0.141822], [0,0,0,0], [9E9, 9E9, 9E9, 9E9, 9E9, 9E9]];
	VAR robtarget Openhole_4594 := [[421.09, -33.31, 177.42], [-0.046058, 0.705605, 0.693041, 0.140338], [0,0,0,0], [9E9, 9E9, 9E9, 9E9, 9E9, 9E9]];
	VAR robtarget Openhole_4595 := [[426.53, -33.08, 178.22], [-0.02879, 0.70652, 0.696316, 0.123059], [0,0,0,0], [9E9, 9E9, 9E9, 9E9, 9E9, 9E9]];
	VAR robtarget Openhole_4596 := [[436.37, -32.09, 179.67], [0.001191, 0.707106, 0.701553, 0.088449], [0,0,0,0], [9E9, 9E9, 9E9, 9E9, 9E9, 9E9]];
	VAR robtarget Openhole_4597 := [[438.84, -31.99, 179.99], [0.009291, 0.707046, 0.70257, 0.079972], [0,0,0,0], [9E9, 9E9, 9E9, 9E9, 9E9, 9E9]];
	VAR robtarget Openhole_4598 := [[439.84, -31.99, 180.12], [0.012701, 0.706993, 0.702933, 0.076712], [0,0,0,0], [9E9, 9E9, 9E9, 9E9, 9E9, 9E9]];
	VAR robtarget Openhole_4599 := [[441.33, -32.04, 180.3], [0.017954, 0.706879, 0.703438, 0.071941], [0,0,0,0], [9E9, 9E9, 9E9, 9E9, 9E9, 9E9]];
	VAR robtarget Openhole_4600 := [[442.32, -32.11, 180.42], [0.021553, 0.706778, 0.703747, 0.068851], [0,0,0,0], [9E9, 9E9, 9E9, 9E9, 9E9, 9E9]];
	VAR robtarget Openhole_4601 := [[442.81, -32.16, 180.48], [0.023404, 0.706719, 0.703891, 0.067363], [0,0,0,0], [9E9, 9E9, 9E9, 9E9, 9E9, 9E9]];
	VAR robtarget Openhole_4602 := [[447.23, -32.82, 181.02], [0.040687, 0.705935, 0.704987, 0.054717], [0,0,0,0], [9E9, 9E9, 9E9, 9E9, 9E9, 9E9]];
	VAR robtarget Openhole_4603 := [[448.21, -32.96, 181.15], [0.044497, 0.705705, 0.705202, 0.051865], [0,0,0,0], [9E9, 9E9, 9E9, 9E9, 9E9, 9E9]];
	VAR robtarget Openhole_4604 := [[448.7, -33.01, 181.21], [0.046347, 0.705586, 0.705311, 0.050369], [0,0,0,0], [9E9, 9E9, 9E9, 9E9, 9E9, 9E9]];
	VAR robtarget Openhole_4605 := [[449.2, -33.05, 181.28], [0.04815, 0.705465, 0.70542, 0.048819], [0,0,0,0], [9E9, 9E9, 9E9, 9E9, 9E9, 9E9]];
	VAR robtarget Openhole_4606 := [[449.69, -33.07, 181.35], [0.049904, 0.705344, 0.705529, 0.047212], [0,0,0,0], [9E9, 9E9, 9E9, 9E9, 9E9, 9E9]];
	VAR robtarget Openhole_4607 := [[450.19, -33.08, 181.41], [0.051605, 0.705221, 0.705638, 0.045549], [0,0,0,0], [9E9, 9E9, 9E9, 9E9, 9E9, 9E9]];
	VAR robtarget Openhole_4608 := [[451.18, -33.03, 181.55], [0.054811, 0.704979, 0.705856, 0.042037], [0,0,0,0], [9E9, 9E9, 9E9, 9E9, 9E9, 9E9]];
	VAR robtarget Openhole_4609 := [[451.67, -32.99, 181.61], [0.056327, 0.70486, 0.705963, 0.040205], [0,0,0,0], [9E9, 9E9, 9E9, 9E9, 9E9, 9E9]];
	VAR robtarget Openhole_4610 := [[452.16, -32.92, 181.68], [0.05777, 0.704743, 0.706068, 0.038313], [0,0,0,0], [9E9, 9E9, 9E9, 9E9, 9E9, 9E9]];
	VAR robtarget Openhole_4611 := [[452.65, -32.84, 181.74], [0.059163, 0.704627, 0.70617, 0.036385], [0,0,0,0], [9E9, 9E9, 9E9, 9E9, 9E9, 9E9]];
	VAR robtarget Openhole_4612 := [[453.63, -32.66, 181.86], [0.06182, 0.704399, 0.706362, 0.032436], [0,0,0,0], [9E9, 9E9, 9E9, 9E9, 9E9, 9E9]];
	VAR robtarget Openhole_4613 := [[460.43, -31.22, 182.6], [0.079731, 0.702597, 0.707093, 0.004397], [0,0,0,0], [9E9, 9E9, 9E9, 9E9, 9E9, 9E9]];
	VAR robtarget Openhole_4614 := [[466.84, -30.31, 183.2], [0.097604, 0.700338, 0.706814, -0.020349], [0,0,0,0], [9E9, 9E9, 9E9, 9E9, 9E9, 9E9]];
	VAR robtarget Openhole_4615 := [[476.26, -29.36, 183.98], [0.124072, 0.696137, 0.704984, -0.054745], [0,0,0,0], [9E9, 9E9, 9E9, 9E9, 9E9, 9E9]];
	VAR robtarget Openhole_4616 := [[470.3, -26.56, 182.82], [0.096355, 0.700511, 0.705716, -0.044331], [0,0,0,0], [9E9, 9E9, 9E9, 9E9, 9E9, 9E9]];
	VAR robtarget Openhole_4617 := [[465.31, -26.64, 182.47], [0.080542, 0.702505, 0.706575, -0.027408], [0,0,0,0], [9E9, 9E9, 9E9, 9E9, 9E9, 9E9]];
	VAR robtarget Openhole_4618 := [[464.81, -26.64, 182.43], [0.078911, 0.70269, 0.706638, -0.025735], [0,0,0,0], [9E9, 9E9, 9E9, 9E9, 9E9, 9E9]];
	VAR robtarget Openhole_4619 := [[463.82, -26.63, 182.36], [0.075631, 0.70305, 0.706752, -0.022389], [0,0,0,0], [9E9, 9E9, 9E9, 9E9, 9E9, 9E9]];
	VAR robtarget Openhole_4620 := [[463.32, -26.64, 182.32], [0.073997, 0.703224, 0.706804, -0.020703], [0,0,0,0], [9E9, 9E9, 9E9, 9E9, 9E9, 9E9]];
	VAR robtarget Openhole_4621 := [[462.82, -26.63, 182.29], [0.072338, 0.703397, 0.70685, -0.019037], [0,0,0,0], [9E9, 9E9, 9E9, 9E9, 9E9, 9E9]];
	VAR robtarget Openhole_4622 := [[459.33, -26.59, 182.03], [0.060645, 0.704501, 0.707069, -0.00734], [0,0,0,0], [9E9, 9E9, 9E9, 9E9, 9E9, 9E9]];
	VAR robtarget Openhole_4623 := [[458.83, -26.59, 181.99], [0.058981, 0.704643, 0.707084, -0.005646], [0,0,0,0], [9E9, 9E9, 9E9, 9E9, 9E9, 9E9]];
	VAR robtarget Openhole_4624 := [[458.33, -26.6, 181.96], [0.057327, 0.704779, 0.707096, -0.003941], [0,0,0,0], [9E9, 9E9, 9E9, 9E9, 9E9, 9E9]];
	VAR robtarget Openhole_4625 := [[457.83, -26.59, 181.92], [0.055649, 0.704914, 0.707103, -0.002255], [0,0,0,0], [9E9, 9E9, 9E9, 9E9, 9E9, 9E9]];
	VAR robtarget Openhole_4626 := [[456.34, -26.58, 181.81], [0.050573, 0.705296, 0.707101, 0.002776], [0,0,0,0], [9E9, 9E9, 9E9, 9E9, 9E9, 9E9]];
	VAR robtarget Openhole_4627 := [[455.34, -26.54, 181.73], [0.047101, 0.705536, 0.707081, 0.00605], [0,0,0,0], [9E9, 9E9, 9E9, 9E9, 9E9, 9E9]];
	VAR robtarget Openhole_4628 := [[454.85, -26.49, 181.7], [0.04527, 0.705656, 0.707066, 0.007582], [0,0,0,0], [9E9, 9E9, 9E9, 9E9, 9E9, 9E9]];
	VAR robtarget Openhole_4629 := [[454.35, -26.44, 181.66], [0.043405, 0.705773, 0.707049, 0.009073], [0,0,0,0], [9E9, 9E9, 9E9, 9E9, 9E9, 9E9]];
	VAR robtarget Openhole_4630 := [[453.86, -26.35, 181.62], [0.041464, 0.70589, 0.707029, 0.010466], [0,0,0,0], [9E9, 9E9, 9E9, 9E9, 9E9, 9E9]];
	VAR robtarget Openhole_4631 := [[453.37, -26.25, 181.58], [0.039477, 0.706004, 0.707008, 0.011796], [0,0,0,0], [9E9, 9E9, 9E9, 9E9, 9E9, 9E9]];
	VAR robtarget Openhole_4632 := [[452.79, -25.92, 181.53], [0.036386, 0.70617, 0.706994, 0.012653], [0,0,0,0], [9E9, 9E9, 9E9, 9E9, 9E9, 9E9]];
	VAR robtarget Openhole_4633 := [[454.94, -24.42, 181.59], [0.038585, 0.706053, 0.707107, 0.000231], [0,0,0,0], [9E9, 9E9, 9E9, 9E9, 9E9, 9E9]];
	VAR robtarget Openhole_4634 := [[455.54, -24.57, 181.63], [0.041128, 0.70591, 0.707106, -0.001297], [0,0,0,0], [9E9, 9E9, 9E9, 9E9, 9E9, 9E9]];
	VAR robtarget Openhole_4635 := [[456.54, -24.66, 181.69], [0.044769, 0.705688, 0.707093, -0.00439], [0,0,0,0], [9E9, 9E9, 9E9, 9E9, 9E9, 9E9]];
	VAR robtarget Openhole_4636 := [[457.04, -24.68, 181.72], [0.046536, 0.705574, 0.707081, -0.005993], [0,0,0,0], [9E9, 9E9, 9E9, 9E9, 9E9, 9E9]];
	VAR robtarget Openhole_4637 := [[460.52, -24.98, 181.94], [0.059174, 0.704626, 0.706907, -0.016804], [0,0,0,0], [9E9, 9E9, 9E9, 9E9, 9E9, 9E9]];
	VAR robtarget Openhole_4638 := [[457.19, -28.45, 182.01], [0.0597, 0.704582, 0.70708, 0.006194], [0,0,0,0], [9E9, 9E9, 9E9, 9E9, 9E9, 9E9]];
	VAR robtarget Openhole_4639 := [[454.2, -28.65, 181.75], [0.050361, 0.705311, 0.706902, 0.017033], [0,0,0,0], [9E9, 9E9, 9E9, 9E9, 9E9, 9E9]];
	VAR robtarget Openhole_4640 := [[453.71, -28.66, 181.71], [0.048722, 0.705426, 0.706858, 0.01877], [0,0,0,0], [9E9, 9E9, 9E9, 9E9, 9E9, 9E9]];
	VAR robtarget Openhole_4641 := [[452.71, -28.67, 181.61], [0.045382, 0.705649, 0.706759, 0.022187], [0,0,0,0], [9E9, 9E9, 9E9, 9E9, 9E9, 9E9]];
	VAR robtarget Openhole_4642 := [[449.23, -28.52, 181.29], [0.033086, 0.706332, 0.706311, 0.033546], [0,0,0,0], [9E9, 9E9, 9E9, 9E9, 9E9, 9E9]];
	VAR robtarget Openhole_4643 := [[448.73, -28.52, 181.25], [0.031367, 0.706411, 0.70623, 0.03521], [0,0,0,0], [9E9, 9E9, 9E9, 9E9, 9E9, 9E9]];
	VAR robtarget Openhole_4644 := [[448.23, -28.52, 181.2], [0.029673, 0.706484, 0.706143, 0.036901], [0,0,0,0], [9E9, 9E9, 9E9, 9E9, 9E9, 9E9]];
	VAR robtarget Openhole_4645 := [[447.24, -28.52, 181.11], [0.026293, 0.706618, 0.705958, 0.040287], [0,0,0,0], [9E9, 9E9, 9E9, 9E9, 9E9, 9E9]];
	VAR robtarget Openhole_4646 := [[444.75, -28.61, 180.88], [0.018106, 0.706875, 0.705408, 0.048985], [0,0,0,0], [9E9, 9E9, 9E9, 9E9, 9E9, 9E9]];
	VAR robtarget Openhole_4647 := [[443.26, -28.67, 180.74], [0.013238, 0.706983, 0.705024, 0.054227], [0,0,0,0], [9E9, 9E9, 9E9, 9E9, 9E9, 9E9]];
	VAR robtarget Openhole_4648 := [[444.55, -31.6, 180.72], [0.027514, 0.706571, 0.704584, 0.05968], [0,0,0,0], [9E9, 9E9, 9E9, 9E9, 9E9, 9E9]];
	VAR robtarget Openhole_4649 := [[445.54, -31.73, 180.84], [0.031305, 0.706413, 0.704822, 0.056793], [0,0,0,0], [9E9, 9E9, 9E9, 9E9, 9E9, 9E9]];
	VAR robtarget Openhole_4650 := [[446.52, -31.9, 180.95], [0.035192, 0.70623, 0.705039, 0.054034], [0,0,0,0], [9E9, 9E9, 9E9, 9E9, 9E9, 9E9]];
	VAR robtarget Openhole_4651 := [[448.49, -32.14, 181.19], [0.042716, 0.705815, 0.705463, 0.048186], [0,0,0,0], [9E9, 9E9, 9E9, 9E9, 9E9, 9E9]];
	VAR robtarget Openhole_4652 := [[448.98, -32.18, 181.26], [0.044539, 0.705703, 0.705566, 0.046652], [0,0,0,0], [9E9, 9E9, 9E9, 9E9, 9E9, 9E9]];
	VAR robtarget Openhole_4653 := [[449.48, -32.21, 181.32], [0.046317, 0.705588, 0.705669, 0.045068], [0,0,0,0], [9E9, 9E9, 9E9, 9E9, 9E9, 9E9]];
	VAR robtarget Openhole_4654 := [[449.97, -32.23, 181.38], [0.048061, 0.705472, 0.705771, 0.043447], [0,0,0,0], [9E9, 9E9, 9E9, 9E9, 9E9, 9E9]];
	VAR robtarget Openhole_4655 := [[450.47, -32.23, 181.44], [0.049739, 0.705355, 0.705873, 0.041757], [0,0,0,0], [9E9, 9E9, 9E9, 9E9, 9E9, 9E9]];
	VAR robtarget Openhole_4656 := [[450.97, -32.22, 181.51], [0.051372, 0.705238, 0.705973, 0.040025], [0,0,0,0], [9E9, 9E9, 9E9, 9E9, 9E9, 9E9]];
	VAR robtarget Openhole_4657 := [[451.46, -32.18, 181.57], [0.052934, 0.705123, 0.706073, 0.038227], [0,0,0,0], [9E9, 9E9, 9E9, 9E9, 9E9, 9E9]];
	VAR robtarget Openhole_4658 := [[451.95, -32.13, 181.63], [0.054445, 0.705008, 0.70617, 0.036388], [0,0,0,0], [9E9, 9E9, 9E9, 9E9, 9E9, 9E9]];
	VAR robtarget Openhole_4659 := [[452.45, -32.07, 181.69], [0.055895, 0.704894, 0.706265, 0.034497], [0,0,0,0], [9E9, 9E9, 9E9, 9E9, 9E9, 9E9]];
	VAR robtarget Openhole_4660 := [[453.43, -31.9, 181.81], [0.058639, 0.704671, 0.706444, 0.030603], [0,0,0,0], [9E9, 9E9, 9E9, 9E9, 9E9, 9E9]];
	VAR robtarget Openhole_4661 := [[452.74, -30.49, 181.68], [0.051617, 0.70522, 0.706544, 0.028216], [0,0,0,0], [9E9, 9E9, 9E9, 9E9, 9E9, 9E9]];
	VAR robtarget Openhole_4662 := [[451.25, -30.57, 181.51], [0.046836, 0.705554, 0.706311, 0.033541], [0,0,0,0], [9E9, 9E9, 9E9, 9E9, 9E9, 9E9]];
	VAR robtarget Openhole_4663 := [[450.76, -30.57, 181.46], [0.045159, 0.705663, 0.706228, 0.03524], [0,0,0,0], [9E9, 9E9, 9E9, 9E9, 9E9, 9E9]];
	VAR robtarget Openhole_4664 := [[450.26, -30.57, 181.4], [0.043457, 0.70577, 0.706143, 0.036911], [0,0,0,0], [9E9, 9E9, 9E9, 9E9, 9E9, 9E9]];
	VAR robtarget Openhole_4665 := [[446.79, -30.31, 181.02], [0.030813, 0.706435, 0.705487, 0.047833], [0,0,0,0], [9E9, 9E9, 9E9, 9E9, 9E9, 9E9]];
	VAR robtarget Openhole_4666 := [[446.79, -30.31, 181.14], [0.03085, 0.706434, 0.705491, 0.047777], [0,0,0,0], [9E9, 9E9, 9E9, 9E9, 9E9, 9E9]];
	VAR robtarget Openhole_4667 := [[450.26, -30.57, 181.52], [0.043508, 0.705767, 0.706145, 0.036867], [0,0,0,0], [9E9, 9E9, 9E9, 9E9, 9E9, 9E9]];
	VAR robtarget Openhole_4668 := [[450.76, -30.57, 181.58], [0.045212, 0.70566, 0.70623, 0.035198], [0,0,0,0], [9E9, 9E9, 9E9, 9E9, 9E9, 9E9]];
	VAR robtarget Openhole_4669 := [[451.25, -30.57, 181.63], [0.046891, 0.70555, 0.706313, 0.033501], [0,0,0,0], [9E9, 9E9, 9E9, 9E9, 9E9, 9E9]];
	VAR robtarget Openhole_4670 := [[452.74, -30.49, 181.8], [0.051677, 0.705216, 0.706545, 0.028182], [0,0,0,0], [9E9, 9E9, 9E9, 9E9, 9E9, 9E9]];
	VAR robtarget Openhole_4671 := [[453.43, -31.9, 181.93], [0.058707, 0.704666, 0.706446, 0.030566], [0,0,0,0], [9E9, 9E9, 9E9, 9E9, 9E9, 9E9]];
	VAR robtarget Openhole_4672 := [[452.45, -32.07, 181.81], [0.055959, 0.704889, 0.706267, 0.034456], [0,0,0,0], [9E9, 9E9, 9E9, 9E9, 9E9, 9E9]];
	VAR robtarget Openhole_4673 := [[451.96, -32.13, 181.75], [0.054508, 0.705003, 0.706172, 0.036345], [0,0,0,0], [9E9, 9E9, 9E9, 9E9, 9E9, 9E9]];
	VAR robtarget Openhole_4674 := [[451.46, -32.18, 181.69], [0.052995, 0.705118, 0.706075, 0.038182], [0,0,0,0], [9E9, 9E9, 9E9, 9E9, 9E9, 9E9]];
	VAR robtarget Openhole_4675 := [[450.97, -32.22, 181.63], [0.051432, 0.705234, 0.705976, 0.039978], [0,0,0,0], [9E9, 9E9, 9E9, 9E9, 9E9, 9E9]];
	VAR robtarget Openhole_4676 := [[450.47, -32.23, 181.56], [0.049797, 0.705351, 0.705876, 0.041708], [0,0,0,0], [9E9, 9E9, 9E9, 9E9, 9E9, 9E9]];
	VAR robtarget Openhole_4677 := [[449.97, -32.23, 181.5], [0.048117, 0.705468, 0.705774, 0.043396], [0,0,0,0], [9E9, 9E9, 9E9, 9E9, 9E9, 9E9]];
	VAR robtarget Openhole_4678 := [[449.48, -32.21, 181.44], [0.046371, 0.705585, 0.705672, 0.045015], [0,0,0,0], [9E9, 9E9, 9E9, 9E9, 9E9, 9E9]];
	VAR robtarget Openhole_4679 := [[448.98, -32.18, 181.38], [0.044591, 0.705699, 0.70557, 0.046598], [0,0,0,0], [9E9, 9E9, 9E9, 9E9, 9E9, 9E9]];
	VAR robtarget Openhole_4680 := [[448.49, -32.14, 181.31], [0.042766, 0.705812, 0.705467, 0.04813], [0,0,0,0], [9E9, 9E9, 9E9, 9E9, 9E9, 9E9]];
	VAR robtarget Openhole_4681 := [[446.52, -31.9, 181.07], [0.035234, 0.706228, 0.705044, 0.053972], [0,0,0,0], [9E9, 9E9, 9E9, 9E9, 9E9, 9E9]];
	VAR robtarget Openhole_4682 := [[445.54, -31.73, 180.96], [0.031342, 0.706412, 0.704828, 0.056728], [0,0,0,0], [9E9, 9E9, 9E9, 9E9, 9E9, 9E9]];
	VAR robtarget Openhole_4683 := [[444.55, -31.6, 180.84], [0.027547, 0.70657, 0.70459, 0.059612], [0,0,0,0], [9E9, 9E9, 9E9, 9E9, 9E9, 9E9]];
	VAR robtarget Openhole_4684 := [[443.26, -28.67, 180.86], [0.013255, 0.706983, 0.705029, 0.054164], [0,0,0,0], [9E9, 9E9, 9E9, 9E9, 9E9, 9E9]];
	VAR robtarget Openhole_4685 := [[444.75, -28.61, 181], [0.018128, 0.706874, 0.705412, 0.048929], [0,0,0,0], [9E9, 9E9, 9E9, 9E9, 9E9, 9E9]];
	VAR robtarget Openhole_4686 := [[447.24, -28.52, 181.23], [0.026325, 0.706617, 0.705961, 0.04024], [0,0,0,0], [9E9, 9E9, 9E9, 9E9, 9E9, 9E9]];
	VAR robtarget Openhole_4687 := [[448.73, -28.52, 181.37], [0.031405, 0.706409, 0.706232, 0.035169], [0,0,0,0], [9E9, 9E9, 9E9, 9E9, 9E9, 9E9]];
	VAR robtarget Openhole_4688 := [[449.23, -28.52, 181.41], [0.033125, 0.70633, 0.706312, 0.033506], [0,0,0,0], [9E9, 9E9, 9E9, 9E9, 9E9, 9E9]];
	VAR robtarget Openhole_4689 := [[452.71, -28.67, 181.73], [0.045435, 0.705646, 0.706759, 0.02216], [0,0,0,0], [9E9, 9E9, 9E9, 9E9, 9E9, 9E9]];
	VAR robtarget Openhole_4690 := [[453.71, -28.66, 181.83], [0.048779, 0.705422, 0.706858, 0.018747], [0,0,0,0], [9E9, 9E9, 9E9, 9E9, 9E9, 9E9]];
	VAR robtarget Openhole_4691 := [[454.2, -28.65, 181.87], [0.050419, 0.705307, 0.706902, 0.017012], [0,0,0,0], [9E9, 9E9, 9E9, 9E9, 9E9, 9E9]];
	VAR robtarget Openhole_4692 := [[457.19, -28.45, 182.13], [0.059769, 0.704576, 0.70708, 0.006185], [0,0,0,0], [9E9, 9E9, 9E9, 9E9, 9E9, 9E9]];
	VAR robtarget Openhole_4693 := [[460.52, -24.98, 182.06], [0.059242, 0.704621, 0.706908, -0.016786], [0,0,0,0], [9E9, 9E9, 9E9, 9E9, 9E9, 9E9]];
	VAR robtarget Openhole_4694 := [[457.04, -24.68, 181.84], [0.04659, 0.70557, 0.707081, -0.005988], [0,0,0,0], [9E9, 9E9, 9E9, 9E9, 9E9, 9E9]];
	VAR robtarget Openhole_4695 := [[456.54, -24.66, 181.81], [0.044821, 0.705685, 0.707093, -0.004386], [0,0,0,0], [9E9, 9E9, 9E9, 9E9, 9E9, 9E9]];
	VAR robtarget Openhole_4696 := [[455.54, -24.57, 181.75], [0.041176, 0.705907, 0.707106, -0.001297], [0,0,0,0], [9E9, 9E9, 9E9, 9E9, 9E9, 9E9]];
	VAR robtarget Openhole_4697 := [[454.94, -24.42, 181.71], [0.03863, 0.706051, 0.707107, 0.00023], [0,0,0,0], [9E9, 9E9, 9E9, 9E9, 9E9, 9E9]];
	VAR robtarget Openhole_4698 := [[452.79, -25.92, 181.65], [0.036429, 0.706168, 0.706994, 0.012637], [0,0,0,0], [9E9, 9E9, 9E9, 9E9, 9E9, 9E9]];
	VAR robtarget Openhole_4699 := [[453.37, -26.25, 181.7], [0.039524, 0.706001, 0.707009, 0.011781], [0,0,0,0], [9E9, 9E9, 9E9, 9E9, 9E9, 9E9]];
	VAR robtarget Openhole_4700 := [[453.86, -26.35, 181.74], [0.041513, 0.705887, 0.70703, 0.010453], [0,0,0,0], [9E9, 9E9, 9E9, 9E9, 9E9, 9E9]];
	VAR robtarget Openhole_4701 := [[454.35, -26.44, 181.78], [0.043455, 0.70577, 0.707049, 0.009061], [0,0,0,0], [9E9, 9E9, 9E9, 9E9, 9E9, 9E9]];
	VAR robtarget Openhole_4702 := [[454.85, -26.49, 181.82], [0.045323, 0.705653, 0.707066, 0.007572], [0,0,0,0], [9E9, 9E9, 9E9, 9E9, 9E9, 9E9]];
	VAR robtarget Openhole_4703 := [[455.34, -26.54, 181.85], [0.047155, 0.705533, 0.707081, 0.006041], [0,0,0,0], [9E9, 9E9, 9E9, 9E9, 9E9, 9E9]];
	VAR robtarget Openhole_4704 := [[456.34, -26.58, 181.93], [0.050632, 0.705292, 0.707101, 0.002771], [0,0,0,0], [9E9, 9E9, 9E9, 9E9, 9E9, 9E9]];
	VAR robtarget Openhole_4705 := [[458.33, -26.6, 182.08], [0.057393, 0.704774, 0.707096, -0.003938], [0,0,0,0], [9E9, 9E9, 9E9, 9E9, 9E9, 9E9]];
	VAR robtarget Openhole_4706 := [[458.83, -26.59, 182.11], [0.059049, 0.704637, 0.707084, -0.005642], [0,0,0,0], [9E9, 9E9, 9E9, 9E9, 9E9, 9E9]];
	VAR robtarget Openhole_4707 := [[459.33, -26.59, 182.15], [0.060714, 0.704495, 0.707069, -0.007334], [0,0,0,0], [9E9, 9E9, 9E9, 9E9, 9E9, 9E9]];
	VAR robtarget Openhole_4708 := [[459.83, -26.6, 182.19], [0.062389, 0.704349, 0.707049, -0.009013], [0,0,0,0], [9E9, 9E9, 9E9, 9E9, 9E9, 9E9]];
	VAR robtarget Openhole_4709 := [[463.32, -26.64, 182.44], [0.07408, 0.703216, 0.706804, -0.020682], [0,0,0,0], [9E9, 9E9, 9E9, 9E9, 9E9, 9E9]];
	VAR robtarget Openhole_4710 := [[463.82, -26.63, 182.48], [0.075716, 0.703041, 0.706753, -0.022366], [0,0,0,0], [9E9, 9E9, 9E9, 9E9, 9E9, 9E9]];
	VAR robtarget Openhole_4711 := [[464.32, -26.64, 182.52], [0.077361, 0.702862, 0.706698, -0.024036], [0,0,0,0], [9E9, 9E9, 9E9, 9E9, 9E9, 9E9]];
	VAR robtarget Openhole_4712 := [[465.31, -26.64, 182.59], [0.080632, 0.702494, 0.706577, -0.02738], [0,0,0,0], [9E9, 9E9, 9E9, 9E9, 9E9, 9E9]];
	VAR robtarget Openhole_4713 := [[465.81, -26.64, 182.63], [0.082252, 0.702307, 0.706509, -0.02906], [0,0,0,0], [9E9, 9E9, 9E9, 9E9, 9E9, 9E9]];
	VAR robtarget Openhole_4714 := [[470.3, -26.56, 182.94], [0.09646, 0.700497, 0.705719, -0.044284], [0,0,0,0], [9E9, 9E9, 9E9, 9E9, 9E9, 9E9]];
	VAR robtarget Openhole_4715 := [[476.26, -29.36, 184.1], [0.124201, 0.696114, 0.704989, -0.054689], [0,0,0,0], [9E9, 9E9, 9E9, 9E9, 9E9, 9E9]];
	VAR robtarget Openhole_4716 := [[466.35, -30.36, 183.28], [0.096307, 0.700518, 0.706865, -0.018472], [0,0,0,0], [9E9, 9E9, 9E9, 9E9, 9E9, 9E9]];
	VAR robtarget Openhole_4717 := [[460.44, -31.22, 182.72], [0.07982, 0.702587, 0.707093, 0.00439], [0,0,0,0], [9E9, 9E9, 9E9, 9E9, 9E9, 9E9]];
	VAR robtarget Openhole_4718 := [[453.63, -32.66, 181.98], [0.061891, 0.704393, 0.706364, 0.032397], [0,0,0,0], [9E9, 9E9, 9E9, 9E9, 9E9, 9E9]];
	VAR robtarget Openhole_4719 := [[452.65, -32.84, 181.86], [0.059231, 0.704622, 0.706172, 0.036342], [0,0,0,0], [9E9, 9E9, 9E9, 9E9, 9E9, 9E9]];
	VAR robtarget Openhole_4720 := [[452.16, -32.92, 181.8], [0.057836, 0.704738, 0.706071, 0.038268], [0,0,0,0], [9E9, 9E9, 9E9, 9E9, 9E9, 9E9]];
	VAR robtarget Openhole_4721 := [[451.67, -32.99, 181.73], [0.056392, 0.704855, 0.705966, 0.040157], [0,0,0,0], [9E9, 9E9, 9E9, 9E9, 9E9, 9E9]];
	VAR robtarget Openhole_4722 := [[451.18, -33.03, 181.67], [0.054875, 0.704974, 0.705859, 0.041987], [0,0,0,0], [9E9, 9E9, 9E9, 9E9, 9E9, 9E9]];
	VAR robtarget Openhole_4723 := [[450.19, -33.08, 181.53], [0.051665, 0.705217, 0.705642, 0.045496], [0,0,0,0], [9E9, 9E9, 9E9, 9E9, 9E9, 9E9]];
	VAR robtarget Openhole_4724 := [[449.69, -33.07, 181.47], [0.049962, 0.705339, 0.705533, 0.047157], [0,0,0,0], [9E9, 9E9, 9E9, 9E9, 9E9, 9E9]];
	VAR robtarget Openhole_4725 := [[449.2, -33.05, 181.4], [0.048207, 0.705462, 0.705423, 0.048762], [0,0,0,0], [9E9, 9E9, 9E9, 9E9, 9E9, 9E9]];
	VAR robtarget Openhole_4726 := [[448.7, -33.01, 181.33], [0.046402, 0.705583, 0.705315, 0.050311], [0,0,0,0], [9E9, 9E9, 9E9, 9E9, 9E9, 9E9]];
	VAR robtarget Openhole_4727 := [[448.21, -32.96, 181.27], [0.044549, 0.705702, 0.705207, 0.051805], [0,0,0,0], [9E9, 9E9, 9E9, 9E9, 9E9, 9E9]];
	VAR robtarget Openhole_4728 := [[447.23, -32.82, 181.14], [0.040735, 0.705932, 0.704991, 0.054654], [0,0,0,0], [9E9, 9E9, 9E9, 9E9, 9E9, 9E9]];
	VAR robtarget Openhole_4729 := [[442.81, -32.16, 180.6], [0.023433, 0.706718, 0.703898, 0.067286], [0,0,0,0], [9E9, 9E9, 9E9, 9E9, 9E9, 9E9]];
	VAR robtarget Openhole_4730 := [[442.32, -32.11, 180.54], [0.02158, 0.706777, 0.703754, 0.068773], [0,0,0,0], [9E9, 9E9, 9E9, 9E9, 9E9, 9E9]];
	VAR robtarget Openhole_4731 := [[441.33, -32.04, 180.42], [0.017976, 0.706878, 0.703446, 0.07186], [0,0,0,0], [9E9, 9E9, 9E9, 9E9, 9E9, 9E9]];
	VAR robtarget Openhole_4732 := [[439.84, -31.99, 180.24], [0.012717, 0.706992, 0.702943, 0.076626], [0,0,0,0], [9E9, 9E9, 9E9, 9E9, 9E9, 9E9]];
	VAR robtarget Openhole_4733 := [[438.85, -31.99, 180.11], [0.009304, 0.707046, 0.70258, 0.079883], [0,0,0,0], [9E9, 9E9, 9E9, 9E9, 9E9, 9E9]];
	VAR robtarget Openhole_4734 := [[434.39, -32.25, 179.52], [-0.004979, 0.707089, 0.700654, 0.095313], [0,0,0,0], [9E9, 9E9, 9E9, 9E9, 9E9, 9E9]];
	VAR robtarget Openhole_4735 := [[426.03, -33.12, 178.26], [-0.030342, 0.706455, 0.696046, 0.124577], [0,0,0,0], [9E9, 9E9, 9E9, 9E9, 9E9, 9E9]];
	VAR robtarget Openhole_4736 := [[420.59, -33.32, 177.47], [-0.04772, 0.705495, 0.692768, 0.14168], [0,0,0,0], [9E9, 9E9, 9E9, 9E9, 9E9, 9E9]];
	VAR robtarget Openhole_4737 := [[420.1, -33.31, 177.4], [-0.049348, 0.705383, 0.692466, 0.143146], [0,0,0,0], [9E9, 9E9, 9E9, 9E9, 9E9, 9E9]];
	VAR robtarget Openhole_4738 := [[413.65, -33.07, 176.6], [-0.070906, 0.703543, 0.688524, 0.161043], [0,0,0,0], [9E9, 9E9, 9E9, 9E9, 9E9, 9E9]];
	VAR robtarget Openhole_4739 := [[411.67, -32.92, 176.39], [-0.077631, 0.702832, 0.687311, 0.166144], [0,0,0,0], [9E9, 9E9, 9E9, 9E9, 9E9, 9E9]];
	VAR robtarget Openhole_4740 := [[404.2, -33.45, 175.16], [-0.098926, 0.700153, 0.681699, 0.187845], [0,0,0,0], [9E9, 9E9, 9E9, 9E9, 9E9, 9E9]];
	VAR robtarget Openhole_4741 := [[411.12, -34.32, 175.8], [-0.074998, 0.703118, 0.685885, 0.171937], [0,0,0,0], [9E9, 9E9, 9E9, 9E9, 9E9, 9E9]];
	VAR robtarget Openhole_4742 := [[417.05, -34.8, 176.52], [-0.054521, 0.705002, 0.689526, 0.156695], [0,0,0,0], [9E9, 9E9, 9E9, 9E9, 9E9, 9E9]];
	VAR robtarget Openhole_4743 := [[422, -34.94, 177.23], [-0.037849, 0.706093, 0.692574, 0.142625], [0,0,0,0], [9E9, 9E9, 9E9, 9E9, 9E9, 9E9]];
	VAR robtarget Openhole_4744 := [[422.49, -34.94, 177.31], [-0.036221, 0.706178, 0.692878, 0.141137], [0,0,0,0], [9E9, 9E9, 9E9, 9E9, 9E9, 9E9]];
	VAR robtarget Openhole_4745 := [[428.41, -34.71, 178.26], [-0.017172, 0.706898, 0.696452, 0.12229], [0,0,0,0], [9E9, 9E9, 9E9, 9E9, 9E9, 9E9]];
	VAR robtarget Openhole_4746 := [[436.29, -34.15, 179.52], [0.007769, 0.707064, 0.700647, 0.095363], [0,0,0,0], [9E9, 9E9, 9E9, 9E9, 9E9, 9E9]];
	VAR robtarget Openhole_4747 := [[437.77, -34.12, 179.74], [0.012741, 0.706992, 0.701301, 0.090426], [0,0,0,0], [9E9, 9E9, 9E9, 9E9, 9E9, 9E9]];
	VAR robtarget Openhole_4748 := [[438.27, -34.12, 179.81], [0.014443, 0.706959, 0.701507, 0.088813], [0,0,0,0], [9E9, 9E9, 9E9, 9E9, 9E9, 9E9]];
	VAR robtarget Openhole_4749 := [[438.76, -34.13, 179.88], [0.016166, 0.706922, 0.701707, 0.087219], [0,0,0,0], [9E9, 9E9, 9E9, 9E9, 9E9, 9E9]];
	VAR robtarget Openhole_4750 := [[439.75, -34.17, 180.02], [0.019696, 0.706832, 0.702087, 0.084105], [0,0,0,0], [9E9, 9E9, 9E9, 9E9, 9E9, 9E9]];
	VAR robtarget Openhole_4751 := [[440.74, -34.25, 180.16], [0.023324, 0.706722, 0.702442, 0.081085], [0,0,0,0], [9E9, 9E9, 9E9, 9E9, 9E9, 9E9]];
	VAR robtarget Openhole_4752 := [[441.73, -34.35, 180.3], [0.027043, 0.706589, 0.702774, 0.078161], [0,0,0,0], [9E9, 9E9, 9E9, 9E9, 9E9, 9E9]];
	VAR robtarget Openhole_4753 := [[443.68, -34.65, 180.57], [0.034746, 0.706253, 0.703366, 0.072634], [0,0,0,0], [9E9, 9E9, 9E9, 9E9, 9E9, 9E9]];
	VAR robtarget Openhole_4754 := [[446.59, -35.25, 180.99], [0.046655, 0.705566, 0.704129, 0.064826], [0,0,0,0], [9E9, 9E9, 9E9, 9E9, 9E9, 9E9]];
	VAR robtarget Openhole_4755 := [[447.57, -35.43, 181.14], [0.050566, 0.705296, 0.704371, 0.062144], [0,0,0,0], [9E9, 9E9, 9E9, 9E9, 9E9, 9E9]];
	VAR robtarget Openhole_4756 := [[448.06, -35.5, 181.22], [0.052466, 0.705158, 0.704494, 0.060729], [0,0,0,0], [9E9, 9E9, 9E9, 9E9, 9E9, 9E9]];
	VAR robtarget Openhole_4757 := [[448.55, -35.55, 181.29], [0.054316, 0.705018, 0.70462, 0.05925], [0,0,0,0], [9E9, 9E9, 9E9, 9E9, 9E9, 9E9]];
	VAR robtarget Openhole_4758 := [[449.04, -35.59, 181.37], [0.056112, 0.704877, 0.704748, 0.057706], [0,0,0,0], [9E9, 9E9, 9E9, 9E9, 9E9, 9E9]];
	VAR robtarget Openhole_4759 := [[449.53, -35.6, 181.45], [0.05783, 0.704738, 0.70488, 0.056078], [0,0,0,0], [9E9, 9E9, 9E9, 9E9, 9E9, 9E9]];
	VAR robtarget Openhole_4760 := [[450.03, -35.58, 181.53], [0.059446, 0.704604, 0.705015, 0.054346], [0,0,0,0], [9E9, 9E9, 9E9, 9E9, 9E9, 9E9]];
	VAR robtarget Openhole_4761 := [[450.52, -35.55, 181.61], [0.060999, 0.704471, 0.705151, 0.052559], [0,0,0,0], [9E9, 9E9, 9E9, 9E9, 9E9, 9E9]];
	VAR robtarget Openhole_4762 := [[451.01, -35.49, 181.68], [0.062473, 0.704342, 0.705286, 0.050707], [0,0,0,0], [9E9, 9E9, 9E9, 9E9, 9E9, 9E9]];
	VAR robtarget Openhole_4763 := [[451.5, -35.42, 181.76], [0.063901, 0.704214, 0.70542, 0.048817], [0,0,0,0], [9E9, 9E9, 9E9, 9E9, 9E9, 9E9]];
	VAR robtarget Openhole_4764 := [[451.98, -35.33, 181.84], [0.065229, 0.704092, 0.705553, 0.046857], [0,0,0,0], [9E9, 9E9, 9E9, 9E9, 9E9, 9E9]];
	VAR robtarget Openhole_4765 := [[452.47, -35.23, 181.91], [0.066518, 0.703971, 0.705682, 0.044869], [0,0,0,0], [9E9, 9E9, 9E9, 9E9, 9E9, 9E9]];
	VAR robtarget Openhole_4766 := [[453.43, -34.99, 182.05], [0.068997, 0.703733, 0.705927, 0.040827], [0,0,0,0], [9E9, 9E9, 9E9, 9E9, 9E9, 9E9]];
	VAR robtarget Openhole_4767 := [[460.14, -33.18, 182.89], [0.08534, 0.701938, 0.707006, 0.011931], [0,0,0,0], [9E9, 9E9, 9E9, 9E9, 9E9, 9E9]];
	VAR robtarget Openhole_4768 := [[461.11, -32.96, 183], [0.0878, 0.701635, 0.707063, 0.007894], [0,0,0,0], [9E9, 9E9, 9E9, 9E9, 9E9, 9E9]];
	VAR robtarget Openhole_4769 := [[460.13, -34.45, 183.02], [0.089493, 0.701421, 0.706922, 0.016186], [0,0,0,0], [9E9, 9E9, 9E9, 9E9, 9E9, 9E9]];
	VAR robtarget Openhole_4770 := [[452.05, -36.86, 181.89], [0.070509, 0.703583, 0.705217, 0.051659], [0,0,0,0], [9E9, 9E9, 9E9, 9E9, 9E9, 9E9]];
	VAR robtarget Openhole_4771 := [[451.58, -36.98, 181.81], [0.069308, 0.703702, 0.705065, 0.053693], [0,0,0,0], [9E9, 9E9, 9E9, 9E9, 9E9, 9E9]];
	VAR robtarget Openhole_4772 := [[451.1, -37.12, 181.73], [0.068148, 0.703815, 0.704906, 0.055749], [0,0,0,0], [9E9, 9E9, 9E9, 9E9, 9E9, 9E9]];
	VAR robtarget Openhole_4773 := [[450.62, -37.23, 181.64], [0.066907, 0.703934, 0.704744, 0.057755], [0,0,0,0], [9E9, 9E9, 9E9, 9E9, 9E9, 9E9]];
	VAR robtarget Openhole_4774 := [[450.15, -37.36, 181.56], [0.065727, 0.704045, 0.704574, 0.059795], [0,0,0,0], [9E9, 9E9, 9E9, 9E9, 9E9, 9E9]];
	VAR robtarget Openhole_4775 := [[449.18, -37.57, 181.39], [0.063127, 0.704283, 0.704229, 0.063728], [0,0,0,0], [9E9, 9E9, 9E9, 9E9, 9E9, 9E9]];
	VAR robtarget Openhole_4776 := [[448.69, -37.57, 181.3], [0.06148, 0.704429, 0.704074, 0.065416], [0,0,0,0], [9E9, 9E9, 9E9, 9E9, 9E9, 9E9]];
	VAR robtarget Openhole_4777 := [[448.2, -37.57, 181.22], [0.059788, 0.704575, 0.70392, 0.067058], [0,0,0,0], [9E9, 9E9, 9E9, 9E9, 9E9, 9E9]];
	VAR robtarget Openhole_4778 := [[447.24, -37.35, 181.05], [0.055804, 0.704901, 0.703674, 0.069593], [0,0,0,0], [9E9, 9E9, 9E9, 9E9, 9E9, 9E9]];
	VAR robtarget Openhole_4779 := [[446.78, -37.17, 180.97], [0.053637, 0.70507, 0.70358, 0.070534], [0,0,0,0], [9E9, 9E9, 9E9, 9E9, 9E9, 9E9]];
	VAR robtarget Openhole_4780 := [[446.31, -37, 180.9], [0.051505, 0.705228, 0.703477, 0.07156], [0,0,0,0], [9E9, 9E9, 9E9, 9E9, 9E9, 9E9]];
	VAR robtarget Openhole_4781 := [[445.84, -36.87, 180.82], [0.049429, 0.705377, 0.70336, 0.072695], [0,0,0,0], [9E9, 9E9, 9E9, 9E9, 9E9, 9E9]];
	VAR robtarget Openhole_4782 := [[443.91, -36.44, 180.51], [0.041435, 0.705892, 0.702818, 0.077763], [0,0,0,0], [9E9, 9E9, 9E9, 9E9, 9E9, 9E9]];
	VAR robtarget Openhole_4783 := [[442.94, -36.26, 180.36], [0.037502, 0.706112, 0.702522, 0.080395], [0,0,0,0], [9E9, 9E9, 9E9, 9E9, 9E9, 9E9]];
	VAR robtarget Openhole_4784 := [[441.96, -36.1, 180.21], [0.033643, 0.706306, 0.702204, 0.083125], [0,0,0,0], [9E9, 9E9, 9E9, 9E9, 9E9, 9E9]];
	VAR robtarget Openhole_4785 := [[440.98, -35.98, 180.06], [0.029867, 0.706476, 0.701862, 0.08596], [0,0,0,0], [9E9, 9E9, 9E9, 9E9, 9E9, 9E9]];
	VAR robtarget Openhole_4786 := [[440, -35.88, 179.91], [0.026193, 0.706621, 0.701495, 0.088909], [0,0,0,0], [9E9, 9E9, 9E9, 9E9, 9E9, 9E9]];
	VAR robtarget Openhole_4787 := [[439.01, -35.82, 179.75], [0.022614, 0.706745, 0.701102, 0.091954], [0,0,0,0], [9E9, 9E9, 9E9, 9E9, 9E9, 9E9]];
	VAR robtarget Openhole_4788 := [[438.02, -35.8, 179.59], [0.019136, 0.706848, 0.700684, 0.095092], [0,0,0,0], [9E9, 9E9, 9E9, 9E9, 9E9, 9E9]];
	VAR robtarget Openhole_4789 := [[437.04, -35.79, 179.44], [0.015741, 0.706932, 0.700241, 0.098297], [0,0,0,0], [9E9, 9E9, 9E9, 9E9, 9E9, 9E9]];
	VAR robtarget Openhole_4790 := [[431.62, -36.07, 178.52], [-0.00184, 0.707104, 0.697431, 0.116576], [0,0,0,0], [9E9, 9E9, 9E9, 9E9, 9E9, 9E9]];
	VAR robtarget Openhole_4791 := [[424.25, -36.48, 177.21], [-0.025421, 0.70665, 0.692969, 0.140691], [0,0,0,0], [9E9, 9E9, 9E9, 9E9, 9E9, 9E9]];
	VAR robtarget Openhole_4792 := [[421.78, -36.5, 176.79], [-0.033554, 0.70631, 0.691413, 0.14815], [0,0,0,0], [9E9, 9E9, 9E9, 9E9, 9E9, 9E9]];
	VAR robtarget Openhole_4793 := [[421.29, -36.5, 176.71], [-0.035202, 0.70623, 0.691101, 0.149599], [0,0,0,0], [9E9, 9E9, 9E9, 9E9, 9E9, 9E9]];
	VAR robtarget Openhole_4794 := [[415.86, -36.27, 175.87], [-0.053729, 0.705063, 0.687676, 0.164628], [0,0,0,0], [9E9, 9E9, 9E9, 9E9, 9E9, 9E9]];
	VAR robtarget Openhole_4795 := [[409.94, -35.68, 175.11], [-0.074431, 0.703178, 0.684001, 0.179285], [0,0,0,0], [9E9, 9E9, 9E9, 9E9, 9E9, 9E9]];
	VAR robtarget Openhole_4796 := [[403.54, -34.74, 174.5], [-0.096982, 0.700425, 0.680153, 0.193368], [0,0,0,0], [9E9, 9E9, 9E9, 9E9, 9E9, 9E9]];
	VAR robtarget Openhole_4797 := [[399.12, -33.92, 174.22], [-0.112479, 0.698103, 0.677603, 0.202126], [0,0,0,0], [9E9, 9E9, 9E9, 9E9, 9E9, 9E9]];
	VAR robtarget Openhole_4798 := [[389.32, -33.92, 172.82], [-0.139889, 0.693131, 0.670282, 0.225215], [0,0,0,0], [9E9, 9E9, 9E9, 9E9, 9E9, 9E9]];
	VAR robtarget Openhole_4799 := [[361.72, -33.92, 172.9], [-0.183051, 0.683002, 0.683002, 0.183051], [0,0,0,0], [9E9, 9E9, 9E9, 9E9, 9E9, 9E9]];
	VAR robtarget Openhole_4800 := [[362.36, -10.64, 186.35], [-0.183051, 0.683002, 0.683002, 0.183051], [0,0,0,0], [9E9, 9E9, 9E9, 9E9, 9E9, 9E9]];
	VAR robtarget Openhole_4801 := [[389.36, -10.64, 186.26], [-0.206187, 0.676378, 0.688882, 0.159504], [0,0,0,0], [9E9, 9E9, 9E9, 9E9, 9E9, 9E9]];
	VAR robtarget Openhole_4802 := [[394.36, -10.64, 185.86], [-0.19413, 0.679936, 0.691798, 0.146342], [0,0,0,0], [9E9, 9E9, 9E9, 9E9, 9E9, 9E9]];
	VAR robtarget Openhole_4803 := [[407.75, -10.06, 185.01], [-0.160712, 0.688601, 0.699027, 0.106588], [0,0,0,0], [9E9, 9E9, 9E9, 9E9, 9E9, 9E9]];
	VAR robtarget Openhole_4804 := [[423.69, -9.33, 183.82], [-0.116054, 0.697518, 0.705012, 0.054394], [0,0,0,0], [9E9, 9E9, 9E9, 9E9, 9E9, 9E9]];
	VAR robtarget Openhole_4805 := [[437.6, -8.31, 182.63], [-0.07466, 0.703154, 0.707092, 0.004618], [0,0,0,0], [9E9, 9E9, 9E9, 9E9, 9E9, 9E9]];
	VAR robtarget Openhole_4806 := [[444.02, -7.49, 182.01], [-0.05595, 0.70489, 0.706825, -0.019959], [0,0,0,0], [9E9, 9E9, 9E9, 9E9, 9E9, 9E9]];
	VAR robtarget Openhole_4807 := [[444.51, -7.43, 181.96], [-0.054478, 0.705005, 0.70677, -0.021836], [0,0,0,0], [9E9, 9E9, 9E9, 9E9, 9E9, 9E9]];
	VAR robtarget Openhole_4808 := [[445.5, -7.33, 181.85], [-0.051467, 0.705231, 0.706645, -0.025537], [0,0,0,0], [9E9, 9E9, 9E9, 9E9, 9E9, 9E9]];
	VAR robtarget Openhole_4809 := [[446.49, -7.27, 181.74], [-0.048333, 0.705453, 0.706506, -0.029136], [0,0,0,0], [9E9, 9E9, 9E9, 9E9, 9E9, 9E9]];
	VAR robtarget Openhole_4810 := [[447.49, -7.25, 181.63], [-0.045029, 0.705672, 0.706356, -0.032582], [0,0,0,0], [9E9, 9E9, 9E9, 9E9, 9E9, 9E9]];
	VAR robtarget Openhole_4811 := [[448.48, -7.26, 181.52], [-0.041617, 0.705881, 0.706194, -0.035923], [0,0,0,0], [9E9, 9E9, 9E9, 9E9, 9E9, 9E9]];
	VAR robtarget Openhole_4812 := [[452.45, -7.48, 181.08], [-0.027343, 0.706578, 0.705433, -0.048627], [0,0,0,0], [9E9, 9E9, 9E9, 9E9, 9E9, 9E9]];
	VAR robtarget Openhole_4813 := [[455.43, -7.61, 180.75], [-0.016721, 0.706909, 0.704706, -0.058215], [0,0,0,0], [9E9, 9E9, 9E9, 9E9, 9E9, 9E9]];
	VAR robtarget Openhole_4814 := [[457.42, -7.57, 180.53], [-0.010077, 0.707035, 0.704112, -0.065009], [0,0,0,0], [9E9, 9E9, 9E9, 9E9, 9E9, 9E9]];
	VAR robtarget Openhole_4815 := [[460.88, -7.27, 180.12], [0.000751, 0.707106, 0.702849, -0.077479], [0,0,0,0], [9E9, 9E9, 9E9, 9E9, 9E9, 9E9]];
	VAR robtarget Openhole_4816 := [[471.17, -5.77, 178.64], [0.030525, 0.706448, 0.697604, -0.115536], [0,0,0,0], [9E9, 9E9, 9E9, 9E9, 9E9, 9E9]];
	VAR robtarget Openhole_4817 := [[474.12, -5.49, 178.19], [0.039424, 0.706007, 0.695859, -0.125617], [0,0,0,0], [9E9, 9E9, 9E9, 9E9, 9E9, 9E9]];
	VAR robtarget Openhole_4818 := [[480.82, -3.88, 176.83], [0.056163, 0.704873, 0.690833, -0.150828], [0,0,0,0], [9E9, 9E9, 9E9, 9E9, 9E9, 9E9]];
	VAR robtarget Openhole_4819 := [[478.84, -3.85, 177.11], [0.04964, 0.705362, 0.692062, -0.145089], [0,0,0,0], [9E9, 9E9, 9E9, 9E9, 9E9, 9E9]];
	VAR robtarget Openhole_4820 := [[478.35, -3.86, 177.19], [0.048028, 0.705474, 0.692369, -0.143616], [0,0,0,0], [9E9, 9E9, 9E9, 9E9, 9E9, 9E9]];
	VAR robtarget Openhole_4821 := [[472.91, -4.06, 178.02], [0.030744, 0.706438, 0.695698, -0.126506], [0,0,0,0], [9E9, 9E9, 9E9, 9E9, 9E9, 9E9]];
	VAR robtarget Openhole_4822 := [[464.07, -4.96, 179.43], [0.003894, 0.707096, 0.70062, -0.09556], [0,0,0,0], [9E9, 9E9, 9E9, 9E9, 9E9, 9E9]];
	VAR robtarget Openhole_4823 := [[459.62, -5.2, 180.05], [-0.010456, 0.707029, 0.702546, -0.080186], [0,0,0,0], [9E9, 9E9, 9E9, 9E9, 9E9, 9E9]];
	VAR robtarget Openhole_4824 := [[459.13, -5.2, 180.12], [-0.012142, 0.707003, 0.702731, -0.078541], [0,0,0,0], [9E9, 9E9, 9E9, 9E9, 9E9, 9E9]];
	VAR robtarget Openhole_4825 := [[458.63, -5.19, 180.18], [-0.013873, 0.706971, 0.702909, -0.076934], [0,0,0,0], [9E9, 9E9, 9E9, 9E9, 9E9, 9E9]];
	VAR robtarget Openhole_4826 := [[454.68, -4.82, 180.69], [-0.028621, 0.706527, 0.704113, -0.064996], [0,0,0,0], [9E9, 9E9, 9E9, 9E9, 9E9, 9E9]];
	VAR robtarget Openhole_4827 := [[450.77, -4.2, 181.22], [-0.04408, 0.705731, 0.705051, -0.053881], [0,0,0,0], [9E9, 9E9, 9E9, 9E9, 9E9, 9E9]];
	VAR robtarget Openhole_4828 := [[449.78, -4.1, 181.36], [-0.047774, 0.705491, 0.705274, -0.050884], [0,0,0,0], [9E9, 9E9, 9E9, 9E9, 9E9, 9E9]];
	VAR robtarget Openhole_4829 := [[448.79, -4.06, 181.5], [-0.051262, 0.705246, 0.705499, -0.047652], [0,0,0,0], [9E9, 9E9, 9E9, 9E9, 9E9, 9E9]];
	VAR robtarget Openhole_4830 := [[448.3, -4.06, 181.57], [-0.052942, 0.705122, 0.705611, -0.045971], [0,0,0,0], [9E9, 9E9, 9E9, 9E9, 9E9, 9E9]];
	VAR robtarget Openhole_4831 := [[447.8, -4.1, 181.64], [-0.054481, 0.705005, 0.705726, -0.044161], [0,0,0,0], [9E9, 9E9, 9E9, 9E9, 9E9, 9E9]];
	VAR robtarget Openhole_4832 := [[447.31, -4.15, 181.71], [-0.055988, 0.704887, 0.705839, -0.042322], [0,0,0,0], [9E9, 9E9, 9E9, 9E9, 9E9, 9E9]];
	VAR robtarget Openhole_4833 := [[446.82, -4.21, 181.78], [-0.057435, 0.70477, 0.70595, -0.040437], [0,0,0,0], [9E9, 9E9, 9E9, 9E9, 9E9, 9E9]];
